C01813=1081.570,6.854,-59.285,174.055,20.252,153.427
C01814=1081.564,6.605,-59.270,174.054,20.250,153.427
C01815=1081.558,6.355,-59.257,174.053,20.248,153.427
C01816=1081.553,6.105,-59.243,174.051,20.245,153.426
C01817=1081.546,5.856,-59.228,174.049,20.243,153.426
C01818=1081.541,5.606,-59.214,174.048,20.241,153.426
C01819=1081.535,5.357,-59.200,174.047,20.239,153.426
C01820=1081.530,5.108,-59.185,174.045,20.237,153.426
C01821=1081.523,4.857,-59.171,174.043,20.235,153.426
C01822=1081.517,4.608,-59.158,174.042,20.233,153.425
C01823=1081.512,4.359,-59.143,174.041,20.231,153.425
C01824=1081.507,4.120,-59.130,174.040,20.229,153.425
C01825=1081.500,3.881,-59.116,174.037,20.226,153.425
C01826=1081.495,3.642,-59.103,174.036,20.224,153.425
C01827=1081.489,3.404,-59.090,174.035,20.222,153.424
C01828=1081.484,3.165,-59.076,174.034,20.220,153.424
C01829=1081.479,2.927,-59.063,174.033,20.218,153.424
C01830=1081.473,2.688,-59.050,174.031,20.216,153.424
C01831=1081.467,2.449,-59.036,174.030,20.214,153.424
C01832=1081.461,2.199,-59.022,174.028,20.211,153.424
C01833=1081.456,1.950,-59.008,174.027,20.209,153.423
C01834=1081.450,1.701,-58.994,174.025,20.207,153.423
C01835=1081.444,1.451,-58.980,174.024,20.205,153.423
C01836=1081.438,1.201,-58.965,174.022,20.203,153.423
C01837=1081.432,0.952,-58.952,174.021,20.201,153.423
C01838=1081.426,0.703,-58.938,174.020,20.198,153.422
C01839=1081.421,0.453,-58.924,174.018,20.196,153.422
C01840=1081.415,0.203,-58.910,174.016,20.194,153.422
C01841=1081.409,-0.047,-58.896,174.015,20.192,153.422
C01842=1081.404,-0.296,-58.882,174.014,20.190,153.422
C01843=1081.398,-0.546,-58.869,174.012,20.188,153.422
C01844=1081.391,-0.822,-58.853,174.010,20.185,153.421
C01845=1081.385,-1.098,-58.837,174.009,20.183,153.421
C01846=1081.378,-1.374,-58.822,174.007,20.180,153.421
C01847=1081.372,-1.650,-58.806,174.006,20.178,153.421
C01848=1081.367,-1.899,-58.792,174.005,20.176,153.421
C01849=1081.360,-2.148,-58.779,174.003,20.173,153.420
C01850=1081.355,-2.398,-58.765,174.001,20.171,153.420
C01851=1081.350,-2.648,-58.751,174.000,20.169,153.420
C01852=1081.344,-2.897,-58.737,173.999,20.167,153.420
C01853=1081.338,-3.146,-58.724,173.997,20.165,153.420
C01854=1081.332,-3.397,-58.710,173.996,20.162,153.420
C01855=1081.326,-3.646,-58.696,173.994,20.160,153.419
C01856=1081.320,-3.896,-58.682,173.993,20.158,153.419
C01857=1081.315,-4.145,-58.669,173.991,20.156,153.419
C01858=1081.308,-4.394,-58.655,173.990,20.154,153.419
C01859=1081.302,-4.645,-58.641,173.988,20.152,153.419
C01860=1081.297,-4.894,-58.627,173.987,20.150,153.419
C01861=1081.290,-5.143,-58.613,173.986,20.148,153.418
C01862=1081.285,-5.392,-58.599,173.984,20.145,153.418
C01863=1081.279,-5.642,-58.586,173.982,20.143,153.418
C01864=1081.273,-5.892,-58.572,173.981,20.141,153.418
C01865=1081.266,-6.141,-58.559,173.980,20.139,153.418
C01866=1081.261,-6.391,-58.545,173.979,20.137,153.418
C01867=1081.255,-6.641,-58.532,173.976,20.135,153.417
C01868=1081.249,-6.890,-58.518,173.975,20.133,153.417
C01869=1081.244,-7.140,-58.504,173.974,20.131,153.417
C01870=1081.237,-7.390,-58.491,173.973,20.129,153.417
C01871=1081.232,-7.639,-58.477,173.971,20.126,153.417
C01872=1081.225,-7.889,-58.464,173.969,20.124,153.417
C01873=1081.220,-8.138,-58.450,173.968,20.122,153.416
C01874=1081.214,-8.388,-58.437,173.967,20.120,153.416
C01875=1081.208,-8.637,-58.423,173.965,20.118,153.416
C01876=1081.202,-8.886,-58.409,173.963,20.116,153.416
C01877=1081.197,-9.136,-58.396,173.962,20.114,153.416
C01878=1081.190,-9.386,-58.382,173.961,20.112,153.416
C01879=1081.184,-9.635,-58.368,173.960,20.110,153.415
C01880=1081.178,-9.885,-58.356,173.957,20.107,153.415
C01881=1081.173,-10.135,-58.342,173.956,20.105,153.415
C01882=1081.167,-10.384,-58.328,173.955,20.103,153.415
C01883=1081.161,-10.634,-58.315,173.954,20.101,153.415
C01884=1081.155,-10.883,-58.301,173.952,20.099,153.415
C01885=1081.150,-11.133,-58.287,173.950,20.097,153.414
C01886=1081.143,-11.382,-58.274,173.949,20.095,153.414
C01887=1081.138,-11.632,-58.261,173.948,20.093,153.414
C01888=1081.132,-11.881,-58.248,173.946,20.091,153.414
C01889=1081.126,-12.131,-58.234,173.945,20.089,153.414
C01890=1081.120,-12.381,-58.220,173.943,20.087,153.414
C01891=1081.114,-12.630,-58.206,173.942,20.085,153.413
C01892=1081.108,-12.880,-58.194,173.940,20.083,153.413
C01893=1081.103,-13.130,-58.180,173.939,20.080,153.413
C01894=1081.097,-13.379,-58.167,173.938,20.078,153.413
C01895=1081.090,-13.628,-58.153,173.936,20.076,153.413
C01896=1081.085,-13.878,-58.139,173.935,20.074,153.413
C01897=1081.079,-14.128,-58.127,173.933,20.072,153.413
C01898=1081.074,-14.377,-58.113,173.932,20.070,153.412
C01899=1081.067,-14.627,-58.100,173.931,20.068,153.412
C01900=1081.062,-14.877,-58.087,173.929,20.065,153.412
C01901=1081.056,-15.126,-58.073,173.928,20.063,153.412
C01902=1081.050,-15.375,-58.060,173.926,20.062,153.412
C01903=1081.044,-15.625,-58.046,173.925,20.060,153.412
C01904=1081.038,-15.875,-58.034,173.924,20.058,153.411
C01905=1081.032,-16.124,-58.020,173.921,20.055,153.411
C01906=1081.027,-16.374,-58.007,173.920,20.053,153.411
C01907=1081.021,-16.624,-57.994,173.919,20.051,153.411
C01908=1081.013,-16.898,-57.979,173.918,20.049,153.411
C01909=1081.008,-17.172,-57.965,173.916,20.047,153.411
C01910=1081.001,-17.447,-57.950,173.914,20.045,153.410
C01911=1080.995,-17.721,-57.936,173.912,20.042,153.410
C01912=1080.989,-17.970,-57.923,173.911,20.040,153.410
C01913=1080.982,-18.220,-57.909,173.910,20.038,153.410
C01914=1080.976,-18.470,-57.897,173.908,20.036,153.410
C01915=1080.971,-18.719,-57.883,173.907,20.034,153.410
C01916=1080.965,-18.968,-57.870,173.905,20.032,153.409
C01917=1080.959,-19.218,-57.857,173.904,20.030,153.409
C01918=1080.953,-19.467,-57.844,173.902,20.028,153.409
C01919=1080.947,-19.717,-57.831,173.901,20.026,153.409
C01920=1080.941,-19.967,-57.817,173.900,20.024,153.409
C01921=1080.935,-20.217,-57.805,173.898,20.021,153.409
C01922=1080.929,-20.466,-57.791,173.897,20.019,153.408
C01923=1080.923,-20.715,-57.778,173.895,20.017,153.408
C01924=1080.918,-20.966,-57.765,173.894,20.015,153.408
C01925=1080.912,-21.215,-57.752,173.892,20.014,153.408
C01926=1080.906,-21.465,-57.739,173.891,20.012,153.408
C01927=1080.899,-21.714,-57.726,173.889,20.009,153.408
C01928=1080.894,-21.964,-57.713,173.888,20.007,153.408
C01929=1080.888,-22.213,-57.700,173.887,20.005,153.407
C01930=1080.882,-22.463,-57.687,173.885,20.003,153.407
C01931=1080.876,-22.713,-57.674,173.884,20.001,153.407
C01932=1080.870,-22.962,-57.661,173.882,19.999,153.407
C01933=1080.865,-23.212,-57.647,173.881,19.997,153.407
C01934=1080.859,-23.462,-57.635,173.879,19.995,153.407
C01935=1080.852,-23.711,-57.621,173.878,19.993,153.406
C01936=1080.847,-23.961,-57.609,173.877,19.991,153.406
C01937=1080.841,-24.210,-57.596,173.875,19.989,153.406
C01938=1080.835,-24.459,-57.583,173.873,19.987,153.406
C01939=1080.830,-24.709,-57.570,173.872,19.985,153.406
C01940=1080.824,-24.959,-57.557,173.871,19.983,153.406
C01941=1080.818,-25.209,-57.545,173.869,19.981,153.406
C01942=1080.811,-25.458,-57.531,173.868,19.979,153.405
C01943=1080.806,-25.708,-57.519,173.866,19.976,153.405
C01944=1080.799,-25.957,-57.505,173.865,19.974,153.405
C01945=1080.794,-26.207,-57.492,173.864,19.972,153.405
C01946=1080.789,-26.457,-57.480,173.862,19.970,153.405
C01947=1080.783,-26.706,-57.467,173.861,19.968,153.405
C01948=1080.777,-26.956,-57.454,173.860,19.967,153.405
C01949=1080.771,-27.205,-57.441,173.857,19.964,153.405
C01950=1080.765,-27.455,-57.428,173.856,19.962,153.404
C01951=1080.759,-27.705,-57.416,173.855,19.960,153.404
C01952=1080.753,-27.954,-57.403,173.854,19.958,153.404
C01953=1080.747,-28.204,-57.390,173.852,19.957,153.404
C01954=1080.741,-28.454,-57.378,173.851,19.955,153.404
C01955=1080.734,-28.703,-57.364,173.849,19.952,153.404
C01956=1080.729,-28.953,-57.352,173.848,19.950,153.404
C01957=1080.723,-29.202,-57.339,173.846,19.948,153.403
C01958=1080.717,-29.451,-57.326,173.845,19.947,153.403
C01959=1080.711,-29.701,-57.314,173.844,19.945,153.403
C01960=1080.705,-29.951,-57.301,173.842,19.943,153.403
C01961=1080.699,-30.201,-57.289,173.840,19.940,153.403
C01962=1080.693,-30.450,-57.275,173.839,19.938,153.403
C01963=1080.687,-30.700,-57.263,173.837,19.937,153.403
C01964=1080.681,-30.950,-57.250,173.836,19.935,153.402
C01965=1080.676,-31.199,-57.238,173.835,19.933,153.402
C01966=1080.669,-31.448,-57.225,173.834,19.931,153.402
C01967=1080.663,-31.698,-57.213,173.832,19.929,153.402
C01968=1080.657,-31.948,-57.200,173.830,19.927,153.402
C01969=1080.651,-32.198,-57.188,173.829,19.925,153.402
C01970=1080.645,-32.447,-57.174,173.827,19.923,153.402
C01971=1080.639,-32.697,-57.162,173.826,19.921,153.401
C01972=1080.633,-32.970,-57.148,173.825,19.919,153.401
C01973=1080.627,-33.244,-57.134,173.823,19.916,153.401
C01974=1080.620,-33.517,-57.121,173.822,19.914,153.401
C01975=1080.613,-33.791,-57.107,173.819,19.912,153.401
C01976=1080.608,-34.041,-57.094,173.818,19.910,153.401
C01977=1080.602,-34.290,-57.082,173.817,19.908,153.401
C01978=1080.596,-34.540,-57.070,173.815,19.906,153.401
C01979=1080.590,-34.790,-57.057,173.814,19.904,153.400
C01980=1080.584,-35.039,-57.044,173.813,19.903,153.400
C01981=1080.578,-35.289,-57.031,173.811,19.901,153.400
C01982=1080.572,-35.539,-57.019,173.809,19.898,153.400
C01983=1080.566,-35.787,-57.007,173.808,19.896,153.400
C01984=1080.560,-36.037,-56.994,173.807,19.894,153.400
C01985=1080.555,-36.287,-56.982,173.805,19.893,153.400
C01986=1080.549,-36.537,-56.969,173.804,19.891,153.399
C01987=1080.543,-36.786,-56.957,173.803,19.889,153.399
C01988=1080.537,-37.036,-56.945,173.802,19.887,153.399
C01989=1080.532,-37.286,-56.932,173.799,19.885,153.399
C01990=1080.525,-37.535,-56.919,173.798,19.883,153.399
C01991=1080.519,-37.784,-56.907,173.797,19.881,153.399
C01992=1080.513,-38.034,-56.895,173.795,19.879,153.399
C01993=1080.507,-38.284,-56.882,173.794,19.877,153.399
C01994=1080.502,-38.534,-56.870,173.793,19.875,153.398
C01995=1080.496,-38.783,-56.857,173.791,19.873,153.398
C01996=1080.490,-39.033,-56.845,173.789,19.871,153.398
C01997=1080.484,-39.282,-56.833,173.788,19.869,153.398
C01998=1080.478,-39.532,-56.820,173.787,19.867,153.398
C01999=1080.472,-39.782,-56.808,173.785,19.866,153.398
C02000=1080.466,-40.031,-56.796,173.784,19.864,153.398
C02001=1080.460,-40.281,-56.784,173.783,19.862,153.398
C02002=1080.454,-40.531,-56.771,173.781,19.860,153.398
C02003=1080.447,-40.780,-56.759,173.779,19.858,153.397
C02004=1080.442,-41.030,-56.747,173.778,19.856,153.397
C02005=1080.436,-41.280,-56.734,173.776,19.854,153.397
C02006=1080.429,-41.529,-56.722,173.775,19.852,153.397
C02007=1080.424,-41.779,-56.710,173.774,19.850,153.397
C02008=1080.418,-42.028,-56.698,173.772,19.849,153.397
C02009=1080.412,-42.278,-56.686,173.771,19.847,153.397
C02010=1080.406,-42.528,-56.673,173.770,19.845,153.397
C02011=1080.401,-42.777,-56.662,173.767,19.843,153.397
C02012=1080.394,-43.027,-56.650,173.766,19.841,153.396
C02013=1080.388,-43.277,-56.637,173.765,19.839,153.396
C02014=1080.382,-43.527,-56.625,173.763,19.837,153.396
C02015=1080.376,-43.776,-56.613,173.762,19.835,153.396
C02016=1080.370,-44.025,-56.600,173.761,19.834,153.396
C02017=1080.364,-44.275,-56.588,173.759,19.832,153.396
C02018=1080.358,-44.524,-56.576,173.758,19.830,153.396
C02019=1080.352,-44.774,-56.564,173.756,19.828,153.396
C02020=1080.347,-45.025,-56.552,173.755,19.826,153.395
C02021=1080.341,-45.274,-56.540,173.753,19.824,153.395
C02022=1080.335,-45.523,-56.528,173.752,19.822,153.395
C02023=1080.329,-45.773,-56.515,173.751,19.820,153.395
C02024=1080.323,-46.022,-56.504,173.749,19.819,153.395
C02025=1080.317,-46.272,-56.491,173.748,19.817,153.395
C02026=1080.311,-46.522,-56.480,173.746,19.815,153.395
C02027=1080.305,-46.771,-56.468,173.745,19.813,153.395
C02028=1080.299,-47.021,-56.455,173.743,19.811,153.395
C02029=1080.293,-47.271,-56.443,173.742,19.809,153.395
C02030=1080.287,-47.520,-56.431,173.740,19.807,153.394
C02031=1080.281,-47.770,-56.420,173.739,19.806,153.394
C02032=1080.275,-48.020,-56.407,173.738,19.804,153.394
C02033=1080.270,-48.269,-56.395,173.736,19.802,153.394
C02034=1080.263,-48.519,-56.383,173.735,19.800,153.394
C02035=1080.258,-48.769,-56.372,173.734,19.798,153.394
C02036=1080.251,-49.042,-56.358,173.731,19.796,153.394
C02037=1080.245,-49.316,-56.344,173.730,19.794,153.394
C02038=1080.238,-49.590,-56.332,173.729,19.792,153.393
C02039=1080.232,-49.864,-56.318,173.727,19.790,153.393
C02040=1080.225,-50.114,-56.307,173.725,19.788,153.393
C02041=1080.220,-50.363,-56.295,173.724,19.786,153.393
C02042=1080.214,-50.613,-56.283,173.722,19.785,153.393
C02043=1080.208,-50.863,-56.271,173.721,19.783,153.393
C02044=1080.202,-51.112,-56.259,173.720,19.781,153.393
C02045=1080.195,-51.362,-56.247,173.718,19.779,153.393
C02046=1080.190,-51.612,-56.236,173.717,19.778,153.393
C02047=1080.184,-51.861,-56.224,173.715,19.776,153.393
C02048=1080.177,-52.111,-56.212,173.713,19.774,153.393
C02049=1080.171,-52.361,-56.200,173.712,19.772,153.393
C02050=1080.165,-52.610,-56.189,173.711,19.770,153.392
C02051=1080.159,-52.860,-56.177,173.709,19.769,153.392
C02052=1080.153,-53.110,-56.165,173.708,19.767,153.392
C02053=1080.147,-53.359,-56.153,173.706,19.765,153.392
C02054=1080.140,-53.609,-56.141,173.705,19.764,153.392
C02055=1080.135,-53.859,-56.130,173.704,19.762,153.392
C02056=1080.129,-54.108,-56.118,173.702,19.760,153.392
C02057=1080.122,-54.358,-56.107,173.701,19.759,153.392
C02058=1080.117,-54.607,-56.094,173.699,19.757,153.392
C02059=1080.110,-54.857,-56.082,173.698,19.755,153.392
C02060=1080.104,-55.107,-56.071,173.696,19.753,153.392
C02061=1080.098,-55.356,-56.060,173.694,19.751,153.392
C02062=1080.092,-55.607,-56.048,173.693,19.750,153.392
C02063=1080.086,-55.855,-56.036,173.692,19.748,153.391
C02064=1080.080,-56.106,-56.025,173.690,19.746,153.391
C02065=1080.074,-56.356,-56.012,173.689,19.744,153.391
C02066=1080.068,-56.604,-56.001,173.687,19.743,153.391
C02067=1080.062,-56.855,-55.990,173.686,19.741,153.391
C02068=1080.056,-57.103,-55.978,173.685,19.739,153.391
C02069=1080.050,-57.354,-55.966,173.683,19.738,153.391
C02070=1080.044,-57.603,-55.954,173.682,19.736,153.391
C02071=1080.038,-57.853,-55.943,173.680,19.734,153.391
C02072=1080.031,-58.103,-55.931,173.678,19.732,153.391
C02073=1080.026,-58.352,-55.920,173.677,19.730,153.391
C02074=1080.019,-58.602,-55.908,173.675,19.729,153.391
C02075=1080.014,-58.851,-55.897,173.674,19.727,153.391
C02076=1080.007,-59.102,-55.886,173.673,19.725,153.390
C02077=1080.002,-59.351,-55.874,173.671,19.724,153.390
C02078=1079.996,-59.601,-55.862,173.670,19.722,153.390
C02079=1079.990,-59.850,-55.851,173.668,19.720,153.390
C02080=1079.983,-60.100,-55.839,173.667,19.719,153.390
C02081=1079.978,-60.349,-55.827,173.665,19.717,153.390
C02082=1079.972,-60.599,-55.816,173.664,19.715,153.390
C02083=1079.966,-60.848,-55.804,173.663,19.714,153.390
C02084=1079.959,-61.099,-55.793,173.661,19.712,153.390
C02085=1079.954,-61.348,-55.782,173.660,19.710,153.390
C02086=1079.948,-61.598,-55.770,173.658,19.708,153.390
C02087=1079.942,-61.847,-55.759,173.656,19.707,153.390
C02088=1079.935,-62.097,-55.747,173.655,19.705,153.389
C02089=1079.930,-62.346,-55.736,173.653,19.703,153.389
C02090=1079.924,-62.597,-55.724,173.652,19.702,153.389
C02091=1079.918,-62.846,-55.713,173.651,19.700,153.389
C02092=1079.912,-63.096,-55.701,173.649,19.698,153.389
C02093=1079.906,-63.346,-55.690,173.648,19.697,153.389
C02094=1079.899,-63.595,-55.679,173.646,19.695,153.389
C02095=1079.894,-63.845,-55.667,173.645,19.693,153.389
C02096=1079.888,-64.095,-55.656,173.644,19.692,153.389
C02097=1079.882,-64.344,-55.644,173.642,19.690,153.389
C02098=1079.875,-64.594,-55.633,173.641,19.688,153.389
C02099=1079.870,-64.844,-55.622,173.639,19.687,153.389
C02100=1079.864,-65.118,-55.609,173.637,19.685,153.389
C02101=1079.856,-65.394,-55.597,173.636,19.683,153.389
C02102=1079.850,-65.669,-55.584,173.634,19.681,153.389
C02103=1079.843,-65.945,-55.572,173.633,19.680,153.389
C02104=1079.837,-66.194,-55.560,173.632,19.678,153.388
C02105=1079.832,-66.444,-55.549,173.630,19.676,153.388
C02106=1079.826,-66.694,-55.538,173.629,19.675,153.388
C02107=1079.820,-66.943,-55.527,173.627,19.672,153.388
C02108=1079.813,-67.193,-55.515,173.625,19.671,153.388
C02109=1079.808,-67.442,-55.504,173.624,19.669,153.388
C02110=1079.802,-67.692,-55.493,173.622,19.668,153.388
C02111=1079.796,-67.942,-55.482,173.621,19.666,153.388
C02112=1079.790,-68.191,-55.470,173.619,19.664,153.388
C02113=1079.784,-68.441,-55.458,173.618,19.663,153.388
C02114=1079.778,-68.691,-55.448,173.616,19.661,153.388
C02115=1079.773,-68.940,-55.437,173.615,19.659,153.388
C02116=1079.766,-69.190,-55.425,173.614,19.658,153.388
C02117=1079.760,-69.439,-55.414,173.612,19.656,153.388
C02118=1079.754,-69.689,-55.403,173.611,19.655,153.388
C02119=1079.748,-69.939,-55.392,173.609,19.653,153.388
C02120=1079.743,-70.189,-55.380,173.608,19.651,153.387
C02121=1079.737,-70.438,-55.369,173.606,19.650,153.387
C02122=1079.731,-70.689,-55.358,173.605,19.648,153.387
C02123=1079.725,-70.938,-55.347,173.604,19.647,153.387
C02124=1079.719,-71.187,-55.336,173.602,19.645,153.387
C02125=1079.713,-71.437,-55.324,173.601,19.643,153.387
C02126=1079.707,-71.687,-55.313,173.599,19.642,153.387
C02127=1079.701,-71.936,-55.303,173.598,19.640,153.387
C02128=1079.695,-72.186,-55.291,173.596,19.639,153.387
C02129=1079.690,-72.436,-55.280,173.595,19.637,153.387
C02130=1079.684,-72.686,-55.269,173.594,19.635,153.387
C02131=1079.678,-72.936,-55.258,173.592,19.634,153.387
C02132=1079.672,-73.185,-55.247,173.591,19.632,153.387
C02133=1079.666,-73.435,-55.236,173.589,19.631,153.387
C02134=1079.660,-73.685,-55.225,173.588,19.629,153.387
C02135=1079.654,-73.934,-55.214,173.585,19.627,153.387
C02136=1079.648,-74.183,-55.202,173.584,19.625,153.387
C02137=1079.643,-74.433,-55.191,173.583,19.624,153.387
C02138=1079.636,-74.683,-55.180,173.581,19.622,153.387
C02139=1079.631,-74.932,-55.169,173.580,19.621,153.387
C02140=1079.624,-75.183,-55.158,173.578,19.619,153.387
C02141=1079.618,-75.432,-55.148,173.577,19.618,153.386
C02142=1079.612,-75.681,-55.137,173.575,19.616,153.386
C02143=1079.606,-75.931,-55.126,173.574,19.615,153.386
C02144=1079.600,-76.181,-55.115,173.572,19.613,153.386
C02145=1079.594,-76.430,-55.104,173.571,19.612,153.386
C02146=1079.588,-76.681,-55.093,173.569,19.610,153.386
C02147=1079.582,-76.930,-55.082,173.568,19.609,153.386
C02148=1079.576,-77.180,-55.071,173.566,19.607,153.386
C02149=1079.570,-77.429,-55.061,173.565,19.606,153.386
C02150=1079.564,-77.679,-55.049,173.563,19.604,153.386
C02151=1079.558,-77.928,-55.039,173.562,19.603,153.386
C02152=1079.552,-78.179,-55.028,173.560,19.601,153.386
C02153=1079.546,-78.429,-55.017,173.559,19.600,153.386
C02154=1079.540,-78.678,-55.006,173.558,19.598,153.386
C02155=1079.535,-78.928,-54.995,173.556,19.597,153.386
C02156=1079.528,-79.177,-54.985,173.555,19.595,153.386
C02157=1079.522,-79.427,-54.974,173.553,19.594,153.386
C02158=1079.516,-79.677,-54.963,173.552,19.592,153.386
C02159=1079.510,-79.926,-54.952,173.550,19.591,153.386
C02160=1079.504,-80.176,-54.941,173.549,19.589,153.386
C02161=1079.497,-80.425,-54.931,173.547,19.588,153.386
C02162=1079.492,-80.675,-54.920,173.546,19.586,153.386
C02163=1079.486,-80.926,-54.909,173.544,19.585,153.386
C02164=1079.479,-81.202,-54.898,173.543,19.584,153.386
C02165=1079.472,-81.480,-54.886,173.541,19.582,153.386
C02166=1079.466,-81.757,-54.873,173.540,19.581,153.386
C02167=1079.458,-82.034,-54.861,173.537,19.579,153.386
C02168=1079.453,-82.284,-54.851,173.537,19.578,153.386
C02169=1079.446,-82.535,-54.840,173.535,19.577,153.386
C02170=1079.440,-82.784,-54.830,173.534,19.575,153.386
C02171=1079.434,-83.033,-54.819,173.532,19.574,153.386
C02172=1079.428,-83.282,-54.809,173.531,19.572,153.386
C02173=1079.422,-83.533,-54.798,173.529,19.571,153.386
C02174=1079.416,-83.783,-54.787,173.528,19.570,153.386
C02175=1079.409,-84.032,-54.777,173.526,19.568,153.386
C02176=1079.403,-84.282,-54.766,173.525,19.567,153.386
C02177=1079.397,-84.532,-54.755,173.523,19.565,153.386
C02178=1079.391,-84.781,-54.745,173.522,19.564,153.386
C02179=1079.385,-85.031,-54.734,173.520,19.562,153.386
C02180=1079.379,-85.281,-54.723,173.518,19.561,153.386
C02181=1079.373,-85.530,-54.713,173.517,19.560,153.386
C02182=1079.367,-85.780,-54.703,173.515,19.558,153.386
C02183=1079.361,-86.030,-54.692,173.514,19.557,153.386
C02184=1079.354,-86.280,-54.681,173.513,19.555,153.386
C02185=1079.349,-86.529,-54.670,173.511,19.554,153.386
C02186=1079.342,-86.779,-54.661,173.509,19.553,153.386
C02187=1079.337,-87.029,-54.650,173.508,19.551,153.386
C02188=1079.330,-87.278,-54.640,173.506,19.550,153.386
C02189=1079.324,-87.529,-54.629,173.505,19.549,153.386
C02190=1079.318,-87.778,-54.618,173.503,19.547,153.386
C02191=1079.312,-88.027,-54.608,173.502,19.546,153.386
C02192=1079.306,-88.277,-54.598,173.500,19.544,153.386
C02193=1079.300,-88.527,-54.587,173.499,19.543,153.386
C02194=1079.294,-88.777,-54.576,173.497,19.542,153.386
C02195=1079.288,-89.027,-54.566,173.496,19.540,153.386
C02196=1079.282,-89.276,-54.556,173.494,19.539,153.386
C02197=1079.276,-89.525,-54.545,173.493,19.537,153.386
C02198=1079.270,-89.775,-54.535,173.491,19.536,153.386
C02199=1079.264,-90.025,-54.524,173.489,19.535,153.386
C02200=1079.258,-90.275,-54.513,173.489,19.534,153.386
C02201=1079.252,-90.525,-54.504,173.487,19.532,153.386
C02202=1079.246,-90.774,-54.493,173.486,19.532,153.386
C02203=1079.240,-91.024,-54.483,173.484,19.530,153.386
C02204=1079.234,-91.274,-54.472,173.483,19.529,153.386
C02205=1079.227,-91.523,-54.462,173.481,19.528,153.386
C02206=1079.221,-91.774,-54.451,173.479,19.526,153.386
C02207=1079.215,-92.023,-54.441,173.478,19.525,153.386
C02208=1079.210,-92.273,-54.431,173.476,19.524,153.386
C02209=1079.204,-92.522,-54.420,173.475,19.522,153.386
C02210=1079.198,-92.772,-54.411,173.473,19.521,153.386
C02211=1079.192,-93.022,-54.400,173.472,19.519,153.386
C02212=1079.185,-93.271,-54.389,173.470,19.518,153.386
C02213=1079.180,-93.521,-54.379,173.469,19.517,153.386
C02214=1079.173,-93.770,-54.369,173.467,19.515,153.386
C02215=1079.167,-94.021,-54.358,173.465,19.514,153.386
C02216=1079.161,-94.270,-54.348,173.464,19.513,153.386
C02217=1079.156,-94.520,-54.338,173.463,19.511,153.386
C02218=1079.149,-94.769,-54.328,173.462,19.511,153.386
C02219=1079.144,-95.019,-54.318,173.460,19.509,153.386
C02220=1079.137,-95.269,-54.307,173.459,19.508,153.386
C02221=1079.132,-95.519,-54.297,173.457,19.507,153.386
C02222=1079.125,-95.768,-54.287,173.456,19.505,153.386
C02223=1079.120,-96.018,-54.277,173.454,19.504,153.386
C02224=1079.114,-96.268,-54.267,173.452,19.503,153.386
C02225=1079.108,-96.517,-54.256,173.451,19.501,153.386
C02226=1079.102,-96.767,-54.247,173.449,19.500,153.386
C02227=1079.096,-97.017,-54.236,173.448,19.499,153.386
C02228=1079.089,-97.297,-54.224,173.446,19.497,153.386
C02229=1079.082,-97.576,-54.213,173.444,19.496,153.386
C02230=1079.076,-97.856,-54.202,173.443,19.495,153.386
C02231=1079.068,-98.136,-54.190,173.442,19.493,153.386
C02232=1079.062,-98.386,-54.180,173.440,19.493,153.387
C02233=1079.056,-98.635,-54.170,173.438,19.491,153.387
C02234=1079.050,-98.885,-54.160,173.437,19.490,153.387
C02235=1079.044,-99.135,-54.150,173.435,19.489,153.387
C02236=1079.038,-99.384,-54.140,173.433,19.488,153.387
C02237=1079.032,-99.634,-54.130,173.432,19.487,153.387
C02238=1079.026,-99.883,-54.120,173.430,19.485,153.387
C02239=1079.020,-100.133,-54.110,173.429,19.484,153.387
C02240=1079.014,-100.383,-54.100,173.427,19.483,153.387
C02241=1079.007,-100.632,-54.090,173.425,19.482,153.387
C02242=1079.001,-100.882,-54.080,173.424,19.480,153.387
C02243=1078.996,-101.132,-54.070,173.423,19.480,153.387
C02244=1078.989,-101.382,-54.059,173.422,19.478,153.387
C02245=1078.983,-101.632,-54.050,173.420,19.477,153.387
C02246=1078.977,-101.882,-54.040,173.418,19.476,153.387
C02247=1078.971,-102.131,-54.029,173.417,19.475,153.387
C02248=1078.965,-102.381,-54.020,173.415,19.473,153.387
C02249=1078.958,-102.631,-54.010,173.413,19.472,153.387
C02250=1078.953,-102.881,-54.000,173.412,19.471,153.387
C02251=1078.946,-103.130,-53.990,173.410,19.470,153.387
C02252=1078.940,-103.380,-53.980,173.409,19.469,153.388
C02253=1078.935,-103.630,-53.970,173.408,19.468,153.387
C02254=1078.928,-103.879,-53.960,173.406,19.467,153.388
C02255=1078.922,-104.129,-53.950,173.405,19.466,153.388
C02256=1078.916,-104.379,-53.941,173.403,19.465,153.388
C02257=1078.911,-104.629,-53.930,173.401,19.464,153.388
C02258=1078.904,-104.878,-53.920,173.400,19.462,153.388
C02259=1078.898,-105.128,-53.911,173.398,19.461,153.388
C02260=1078.892,-105.378,-53.901,173.396,19.460,153.388
C02261=1078.886,-105.628,-53.891,173.395,19.459,153.388
C02262=1078.880,-105.877,-53.881,173.394,19.458,153.388
C02263=1078.874,-106.127,-53.871,173.392,19.457,153.388
C02264=1078.867,-106.376,-53.861,173.391,19.456,153.388
C02265=1078.861,-106.626,-53.852,173.389,19.455,153.388
C02266=1078.856,-106.876,-53.842,173.388,19.454,153.388
C02267=1078.850,-107.126,-53.832,173.386,19.452,153.388
C02268=1078.843,-107.375,-53.822,173.384,19.451,153.388
C02269=1078.837,-107.625,-53.812,173.383,19.450,153.389
C02270=1078.831,-107.875,-53.803,173.382,19.449,153.389
C02271=1078.825,-108.125,-53.793,173.380,19.448,153.389
C02272=1078.819,-108.374,-53.784,173.379,19.447,153.389
C02273=1078.813,-108.625,-53.773,173.377,19.447,153.389
C02274=1078.807,-108.874,-53.763,173.375,19.445,153.389
C02275=1078.800,-109.124,-53.754,173.374,19.444,153.389
C02276=1078.794,-109.373,-53.744,173.372,19.443,153.389
C02277=1078.788,-109.623,-53.734,173.370,19.442,153.389
C02278=1078.782,-109.873,-53.725,173.370,19.441,153.389
C02279=1078.776,-110.123,-53.715,173.368,19.440,153.389
C02280=1078.770,-110.373,-53.706,173.366,19.439,153.389
C02281=1078.763,-110.622,-53.696,173.364,19.438,153.389
C02282=1078.757,-110.872,-53.687,173.363,19.437,153.390
C02283=1078.751,-111.121,-53.677,173.361,19.436,153.390
C02284=1078.745,-111.370,-53.667,173.360,19.435,153.390
C02285=1078.740,-111.621,-53.657,173.359,19.434,153.390
C02286=1078.734,-111.870,-53.647,173.357,19.433,153.390
C02287=1078.727,-112.120,-53.638,173.355,19.432,153.390
C02288=1078.721,-112.370,-53.628,173.354,19.431,153.390
C02289=1078.715,-112.620,-53.619,173.352,19.430,153.390
C02290=1078.709,-112.870,-53.609,173.350,19.429,153.390
C02291=1078.703,-113.119,-53.600,173.349,19.428,153.390
C02292=1078.696,-113.396,-53.589,173.347,19.427,153.390
C02293=1078.689,-113.673,-53.579,173.346,19.426,153.390
C02294=1078.682,-113.950,-53.568,173.344,19.425,153.391
C02295=1078.676,-114.227,-53.557,173.342,19.424,153.391
C02296=1078.670,-114.476,-53.548,173.340,19.423,153.391
C02297=1078.664,-114.726,-53.538,173.340,19.422,153.391
C02298=1078.658,-114.975,-53.529,173.338,19.421,153.391
C02299=1078.652,-115.225,-53.519,173.336,19.420,153.391
C02300=1078.645,-115.475,-53.509,173.334,19.419,153.391
C02301=1078.639,-115.724,-53.501,173.333,19.418,153.391
C02302=1078.632,-115.974,-53.491,173.331,19.417,153.391
C02303=1078.626,-116.224,-53.481,173.330,19.416,153.391
C02304=1078.620,-116.474,-53.472,173.329,19.415,153.391
C02305=1078.614,-116.724,-53.462,173.327,19.415,153.392
C02306=1078.608,-116.973,-53.453,173.325,19.414,153.392
C02307=1078.602,-117.222,-53.443,173.323,19.413,153.392
C02308=1078.596,-117.472,-53.434,173.322,19.412,153.392
C02309=1078.590,-117.723,-53.425,173.321,19.411,153.392
C02310=1078.584,-117.973,-53.415,173.319,19.410,153.392
C02311=1078.578,-118.222,-53.406,173.318,19.409,153.392
C02312=1078.572,-118.472,-53.396,173.316,19.408,153.392
C02313=1078.565,-118.722,-53.387,173.314,19.407,153.392
C02314=1078.559,-118.972,-53.377,173.312,19.406,153.393
C02315=1078.553,-119.220,-53.369,173.312,19.406,153.393
C02316=1078.547,-119.470,-53.359,173.310,19.405,153.393
C02317=1078.541,-119.720,-53.349,173.308,19.404,153.393
C02318=1078.535,-119.971,-53.341,173.306,19.403,153.393
C02319=1078.529,-120.220,-53.331,173.305,19.402,153.393
C02320=1078.522,-120.470,-53.322,173.303,19.401,153.393
C02321=1078.516,-120.720,-53.312,173.302,19.401,153.393
C02322=1078.511,-120.969,-53.303,173.300,19.400,153.393
C02323=1078.504,-121.218,-53.294,173.299,19.399,153.394
C02324=1078.498,-121.469,-53.285,173.297,19.398,153.394
C02325=1078.492,-121.719,-53.275,173.295,19.397,153.394
C02326=1078.485,-121.969,-53.266,173.294,19.396,153.394
C02327=1078.479,-122.218,-53.256,173.293,19.395,153.394
C02328=1078.474,-122.467,-53.247,173.291,19.394,153.394
C02329=1078.468,-122.718,-53.238,173.289,19.394,153.394
C02330=1078.461,-122.967,-53.229,173.287,19.393,153.394
C02331=1078.455,-123.217,-53.220,173.286,19.393,153.395
C02332=1078.449,-123.467,-53.210,173.285,19.392,153.395
C02333=1078.442,-123.717,-53.200,173.283,19.391,153.395
C02334=1078.437,-123.966,-53.192,173.281,19.390,153.395
C02335=1078.430,-124.216,-53.183,173.280,19.389,153.395
C02336=1078.424,-124.466,-53.173,173.279,19.388,153.395
C02337=1078.418,-124.715,-53.164,173.277,19.387,153.395
C02338=1078.412,-124.966,-53.155,173.275,19.387,153.395
C02339=1078.406,-125.215,-53.146,173.273,19.386,153.396
C02340=1078.400,-125.464,-53.137,173.272,19.385,153.396
C02341=1078.394,-125.715,-53.128,173.271,19.384,153.396
C02342=1078.388,-125.965,-53.118,173.269,19.383,153.396
C02343=1078.381,-126.214,-53.109,173.267,19.383,153.396
C02344=1078.375,-126.463,-53.100,173.265,19.382,153.396
C02345=1078.369,-126.714,-53.091,173.264,19.381,153.396
C02346=1078.363,-126.964,-53.082,173.263,19.381,153.396
C02347=1078.356,-127.213,-53.073,173.261,19.380,153.397
C02348=1078.350,-127.463,-53.064,173.259,19.379,153.397
C02349=1078.344,-127.713,-53.054,173.257,19.378,153.397
C02350=1078.338,-127.964,-53.046,173.257,19.378,153.397
C02351=1078.334,-128.214,-53.037,173.255,19.376,153.397
C02352=1078.332,-128.468,-53.025,173.254,19.374,153.397
C02353=1078.334,-128.722,-53.012,173.253,19.371,153.396
C02354=1078.338,-128.975,-53.000,173.253,19.367,153.396
C02355=1078.346,-129.226,-52.986,173.253,19.362,153.395
C02356=1077.949,-129.248,-53.132,173.208,19.486,153.425
C02357=1077.941,-128.998,-53.147,173.209,19.491,153.426
C02358=1077.936,-128.745,-53.159,173.209,19.496,153.427
C02359=1077.935,-128.490,-53.172,173.210,19.499,153.427
C02360=1077.936,-128.235,-53.183,173.211,19.501,153.428
C02361=1077.940,-127.986,-53.193,173.211,19.502,153.428
C02362=1077.946,-127.735,-53.202,173.213,19.503,153.428
C02363=1077.952,-127.485,-53.211,173.215,19.504,153.428
C02364=1077.959,-127.235,-53.220,173.217,19.505,153.427
C02365=1077.965,-126.986,-53.229,173.218,19.506,153.427
C02366=1077.971,-126.735,-53.238,173.219,19.506,153.427
C02367=1077.977,-126.486,-53.247,173.221,19.507,153.427
C02368=1077.983,-126.237,-53.256,173.223,19.508,153.427
C02369=1077.989,-125.986,-53.265,173.224,19.509,153.427
C02370=1077.995,-125.736,-53.275,173.226,19.509,153.427
C02371=1078.002,-125.487,-53.284,173.227,19.510,153.427
C02372=1078.008,-125.237,-53.292,173.229,19.511,153.426
C02373=1078.014,-124.987,-53.302,173.231,19.512,153.426
C02374=1078.020,-124.738,-53.311,173.232,19.513,153.426
C02375=1078.027,-124.488,-53.320,173.234,19.514,153.426
C02376=1078.033,-124.238,-53.329,173.235,19.514,153.426
C02377=1078.039,-123.988,-53.339,173.237,19.514,153.426
C02378=1078.045,-123.739,-53.348,173.239,19.515,153.426
C02379=1078.051,-123.489,-53.358,173.240,19.516,153.425
C02380=1078.057,-123.239,-53.366,173.242,19.517,153.425
C02381=1078.063,-122.989,-53.375,173.243,19.518,153.425
C02382=1078.070,-122.739,-53.385,173.245,19.519,153.425
C02383=1078.075,-122.490,-53.394,173.246,19.520,153.425
C02384=1078.081,-122.240,-53.404,173.248,19.521,153.425
C02385=1078.087,-121.990,-53.413,173.250,19.522,153.425
C02386=1078.094,-121.740,-53.422,173.251,19.522,153.425
C02387=1078.100,-121.491,-53.431,173.252,19.523,153.425
C02388=1078.106,-121.241,-53.441,173.254,19.524,153.425
C02389=1078.112,-120.992,-53.450,173.256,19.525,153.424
C02390=1078.118,-120.742,-53.460,173.257,19.526,153.424
C02391=1078.124,-120.492,-53.468,173.259,19.527,153.424
C02392=1078.130,-120.242,-53.478,173.260,19.527,153.424
C02393=1078.137,-119.992,-53.487,173.262,19.528,153.424
C02394=1078.143,-119.742,-53.496,173.263,19.529,153.424
C02395=1078.150,-119.493,-53.506,173.265,19.530,153.424
C02396=1078.155,-119.244,-53.515,173.267,19.531,153.424
C02397=1078.161,-118.994,-53.525,173.268,19.532,153.424
C02398=1078.167,-118.743,-53.534,173.269,19.533,153.423
C02399=1078.173,-118.494,-53.543,173.271,19.534,153.423
C02400=1078.179,-118.244,-53.553,173.273,19.534,153.423
C02401=1078.186,-117.994,-53.562,173.275,19.535,153.423
C02402=1078.192,-117.744,-53.572,173.276,19.536,153.423
C02403=1078.199,-117.495,-53.581,173.277,19.537,153.423
C02404=1078.204,-117.246,-53.590,173.279,19.538,153.423
C02405=1078.210,-116.996,-53.600,173.281,19.539,153.423
C02406=1078.217,-116.746,-53.609,173.282,19.540,153.423
C02407=1078.223,-116.496,-53.619,173.284,19.541,153.422
C02408=1078.229,-116.246,-53.628,173.286,19.542,153.422
C02409=1078.235,-115.997,-53.638,173.287,19.542,153.422
C02410=1078.241,-115.747,-53.648,173.288,19.544,153.422
C02411=1078.247,-115.497,-53.657,173.290,19.545,153.422
C02412=1078.254,-115.247,-53.667,173.292,19.545,153.422
C02413=1078.260,-114.997,-53.676,173.293,19.546,153.422
C02414=1078.266,-114.747,-53.685,173.295,19.547,153.422
C02415=1078.271,-114.498,-53.694,173.297,19.548,153.422
C02416=1078.277,-114.248,-53.704,173.298,19.549,153.422
C02417=1078.284,-113.971,-53.715,173.299,19.550,153.421
C02418=1078.291,-113.695,-53.725,173.302,19.552,153.421
C02419=1078.298,-113.418,-53.736,173.303,19.553,153.421
C02420=1078.305,-113.141,-53.746,173.305,19.554,153.421
C02421=1078.311,-112.891,-53.756,173.306,19.554,153.421
C02422=1078.317,-112.641,-53.766,173.308,19.555,153.421
C02423=1078.323,-112.391,-53.775,173.309,19.557,153.421
C02424=1078.329,-112.142,-53.785,173.311,19.558,153.421
C02425=1078.335,-111.892,-53.794,173.312,19.558,153.421
C02426=1078.342,-111.642,-53.804,173.314,19.559,153.421
C02427=1078.348,-111.393,-53.814,173.316,19.560,153.421
C02428=1078.354,-111.143,-53.824,173.317,19.562,153.421
C02429=1078.360,-110.893,-53.833,173.318,19.562,153.421
C02430=1078.366,-110.643,-53.843,173.320,19.563,153.420
C02431=1078.372,-110.393,-53.853,173.322,19.564,153.420
C02432=1078.378,-110.143,-53.863,173.323,19.566,153.420
C02433=1078.384,-109.894,-53.872,173.325,19.567,153.420
C02434=1078.390,-109.644,-53.882,173.327,19.568,153.420
C02435=1078.397,-109.394,-53.891,173.328,19.569,153.420
C02436=1078.403,-109.144,-53.901,173.329,19.570,153.420
C02437=1078.409,-108.895,-53.911,173.331,19.571,153.420
C02438=1078.415,-108.645,-53.921,173.332,19.572,153.420
C02439=1078.422,-108.396,-53.930,173.334,19.573,153.420
C02440=1078.428,-108.146,-53.940,173.336,19.574,153.420
C02441=1078.433,-107.896,-53.950,173.337,19.575,153.420
C02442=1078.439,-107.646,-53.960,173.339,19.576,153.419
C02443=1078.446,-107.397,-53.970,173.340,19.577,153.420
C02444=1078.452,-107.147,-53.979,173.341,19.578,153.419
C02445=1078.458,-106.897,-53.989,173.343,19.579,153.419
C02446=1078.464,-106.647,-53.999,173.345,19.580,153.419
C02447=1078.469,-106.398,-54.008,173.346,19.581,153.419
C02448=1078.476,-106.149,-54.019,173.348,19.583,153.419
C02449=1078.482,-105.899,-54.028,173.349,19.584,153.419
C02450=1078.488,-105.649,-54.038,173.351,19.585,153.419
C02451=1078.493,-105.399,-54.048,173.353,19.586,153.419
C02452=1078.500,-105.149,-54.058,173.354,19.587,153.419
C02453=1078.506,-104.900,-54.068,173.355,19.588,153.419
C02454=1078.512,-104.650,-54.077,173.357,19.589,153.419
C02455=1078.518,-104.400,-54.087,173.358,19.590,153.419
C02456=1078.525,-104.150,-54.097,173.360,19.591,153.419
C02457=1078.531,-103.900,-54.108,173.362,19.592,153.419
C02458=1078.537,-103.651,-54.117,173.363,19.594,153.419
C02459=1078.543,-103.401,-54.127,173.365,19.595,153.419
C02460=1078.549,-103.151,-54.137,173.367,19.596,153.418
C02461=1078.555,-102.902,-54.147,173.368,19.597,153.419
C02462=1078.561,-102.652,-54.157,173.370,19.598,153.418
C02463=1078.567,-102.402,-54.167,173.370,19.599,153.418
C02464=1078.573,-102.152,-54.177,173.372,19.600,153.418
C02465=1078.580,-101.903,-54.187,173.374,19.602,153.418
C02466=1078.586,-101.653,-54.196,173.375,19.603,153.418
C02467=1078.591,-101.403,-54.207,173.377,19.604,153.418
C02468=1078.598,-101.154,-54.217,173.378,19.605,153.418
C02469=1078.604,-100.904,-54.226,173.380,19.607,153.418
C02470=1078.610,-100.654,-54.237,173.382,19.608,153.418
C02471=1078.616,-100.404,-54.247,173.383,19.609,153.418
C02472=1078.622,-100.155,-54.256,173.385,19.610,153.418
C02473=1078.628,-99.905,-54.267,173.386,19.611,153.418
C02474=1078.634,-99.655,-54.277,173.387,19.612,153.418
C02475=1078.640,-99.406,-54.286,173.389,19.613,153.418
C02476=1078.647,-99.156,-54.297,173.390,19.614,153.418
C02477=1078.652,-98.906,-54.307,173.392,19.616,153.418
C02478=1078.659,-98.656,-54.318,173.394,19.617,153.418
C02479=1078.665,-98.407,-54.327,173.395,19.618,153.418
C02480=1078.671,-98.156,-54.337,173.397,19.619,153.418
C02481=1078.677,-97.877,-54.349,173.398,19.621,153.418
C02482=1078.685,-97.597,-54.361,173.400,19.622,153.418
C02483=1078.691,-97.317,-54.371,173.401,19.623,153.418
C02484=1078.698,-97.038,-54.383,173.404,19.625,153.418
C02485=1078.703,-96.789,-54.394,173.405,19.626,153.417
C02486=1078.710,-96.539,-54.403,173.406,19.627,153.418
C02487=1078.716,-96.288,-54.414,173.408,19.629,153.418
C02488=1078.722,-96.039,-54.424,173.409,19.630,153.417
C02489=1078.728,-95.789,-54.434,173.411,19.631,153.417
C02490=1078.734,-95.539,-54.444,173.412,19.633,153.417
C02491=1078.740,-95.289,-54.455,173.414,19.634,153.417
C02492=1078.746,-95.040,-54.465,173.415,19.635,153.417
C02493=1078.751,-94.790,-54.475,173.417,19.636,153.417
C02494=1078.758,-94.541,-54.485,173.419,19.637,153.417
C02495=1078.763,-94.291,-54.495,173.420,19.639,153.417
C02496=1078.770,-94.042,-54.506,173.422,19.640,153.417
C02497=1078.775,-93.791,-54.516,173.423,19.642,153.417
C02498=1078.782,-93.542,-54.526,173.425,19.643,153.417
C02499=1078.788,-93.291,-54.537,173.426,19.644,153.417
C02500=1078.794,-93.042,-54.547,173.428,19.646,153.417
C02501=1078.800,-92.793,-54.558,173.429,19.647,153.417
C02502=1078.806,-92.543,-54.567,173.431,19.648,153.417
C02503=1078.812,-92.294,-54.578,173.432,19.649,153.417
C02504=1078.817,-92.043,-54.588,173.433,19.651,153.417
C02505=1078.824,-91.794,-54.599,173.435,19.652,153.417
C02506=1078.829,-91.544,-54.609,173.436,19.653,153.417
C02507=1078.836,-91.294,-54.620,173.438,19.655,153.417
C02508=1078.842,-91.045,-54.630,173.439,19.656,153.417
C02509=1078.848,-90.795,-54.640,173.441,19.657,153.417
C02510=1078.854,-90.545,-54.651,173.442,19.659,153.417
C02511=1078.860,-90.296,-54.660,173.444,19.660,153.417
C02512=1078.866,-90.046,-54.671,173.445,19.662,153.417
C02513=1078.872,-89.796,-54.683,173.447,19.663,153.417
C02514=1078.878,-89.546,-54.692,173.449,19.664,153.417
C02515=1078.884,-89.297,-54.703,173.450,19.666,153.417
C02516=1078.891,-89.048,-54.713,173.452,19.667,153.417
C02517=1078.896,-88.797,-54.723,173.453,19.668,153.417
C02518=1078.902,-88.548,-54.734,173.455,19.669,153.417
C02519=1078.909,-88.298,-54.745,173.456,19.671,153.417
C02520=1078.914,-88.048,-54.755,173.458,19.672,153.417
C02521=1078.921,-87.799,-54.765,173.459,19.674,153.417
C02522=1078.926,-87.549,-54.776,173.461,19.675,153.417
C02523=1078.933,-87.298,-54.787,173.462,19.676,153.417
C02524=1078.939,-87.049,-54.797,173.464,19.678,153.417
C02525=1078.945,-86.800,-54.808,173.465,19.679,153.417
C02526=1078.951,-86.550,-54.818,173.467,19.681,153.417
C02527=1078.957,-86.301,-54.828,173.469,19.682,153.417
C02528=1078.963,-86.050,-54.840,173.469,19.683,153.417
C02529=1078.969,-85.801,-54.850,173.471,19.684,153.417
C02530=1078.975,-85.551,-54.860,173.472,19.686,153.417
C02531=1078.981,-85.302,-54.870,173.474,19.687,153.417
C02532=1078.988,-85.052,-54.882,173.475,19.689,153.417
C02533=1078.993,-84.802,-54.892,173.477,19.690,153.417
C02534=1079.000,-84.552,-54.902,173.478,19.691,153.417
C02535=1079.005,-84.303,-54.913,173.480,19.693,153.417
C02536=1079.012,-84.053,-54.924,173.481,19.694,153.417
C02537=1079.018,-83.804,-54.934,173.483,19.696,153.417
C02538=1079.024,-83.554,-54.945,173.484,19.697,153.417
C02539=1079.029,-83.304,-54.955,173.486,19.699,153.417
C02540=1079.036,-83.054,-54.966,173.487,19.700,153.417
C02541=1079.042,-82.805,-54.977,173.489,19.701,153.417
C02542=1079.048,-82.555,-54.988,173.490,19.703,153.417
C02543=1079.055,-82.305,-54.999,173.492,19.704,153.417
C02544=1079.061,-82.056,-55.009,173.493,19.706,153.417
C02545=1079.068,-81.778,-55.021,173.495,19.707,153.417
C02546=1079.074,-81.500,-55.032,173.497,19.709,153.417
C02547=1079.081,-81.223,-55.045,173.499,19.710,153.417
C02548=1079.088,-80.945,-55.056,173.500,19.712,153.417
C02549=1079.094,-80.696,-55.067,173.502,19.713,153.417
C02550=1079.100,-80.446,-55.078,173.503,19.715,153.417
C02551=1079.106,-80.196,-55.089,173.505,19.716,153.417
C02552=1079.113,-79.947,-55.099,173.506,19.718,153.417
C02553=1079.118,-79.697,-55.110,173.508,19.719,153.417
C02554=1079.125,-79.447,-55.121,173.509,19.721,153.417
C02555=1079.130,-79.198,-55.132,173.511,19.722,153.418
C02556=1079.136,-78.948,-55.143,173.512,19.724,153.418
C02557=1079.143,-78.699,-55.153,173.514,19.725,153.418
C02558=1079.149,-78.448,-55.164,173.515,19.727,153.418
C02559=1079.154,-78.199,-55.175,173.517,19.728,153.418
C02560=1079.160,-77.949,-55.186,173.518,19.730,153.418
C02561=1079.166,-77.699,-55.197,173.519,19.731,153.418
C02562=1079.172,-77.450,-55.208,173.521,19.733,153.418
C02563=1079.178,-77.200,-55.219,173.522,19.734,153.418
C02564=1079.185,-76.950,-55.229,173.524,19.736,153.418
C02565=1079.191,-76.701,-55.240,173.525,19.737,153.418
C02566=1079.197,-76.451,-55.251,173.527,19.739,153.418
C02567=1079.202,-76.202,-55.262,173.528,19.740,153.418
C02568=1079.209,-75.951,-55.273,173.530,19.742,153.418
C02569=1079.214,-75.702,-55.284,173.531,19.743,153.418
C02570=1079.220,-75.453,-55.295,173.533,19.745,153.418
C02571=1079.226,-75.202,-55.306,173.534,19.747,153.418
C02572=1079.232,-74.953,-55.317,173.536,19.748,153.418
C02573=1079.239,-74.703,-55.328,173.537,19.750,153.418
C02574=1079.245,-74.453,-55.339,173.539,19.751,153.418
C02575=1079.251,-74.204,-55.350,173.540,19.753,153.418
C02576=1079.257,-73.954,-55.361,173.542,19.754,153.418
C02577=1079.263,-73.704,-55.372,173.543,19.756,153.418
C02578=1079.269,-73.455,-55.383,173.544,19.757,153.418
C02579=1079.275,-73.206,-55.394,173.546,19.759,153.418
C02580=1079.280,-72.955,-55.406,173.547,19.761,153.418
C02581=1079.286,-72.706,-55.417,173.549,19.762,153.418
C02582=1079.292,-72.456,-55.428,173.550,19.764,153.418
C02583=1079.298,-72.206,-55.439,173.551,19.766,153.419
C02584=1079.304,-71.957,-55.450,173.553,19.767,153.419
C02585=1079.309,-71.707,-55.461,173.554,19.769,153.419
C02586=1079.316,-71.457,-55.472,173.557,19.770,153.419
C02587=1079.322,-71.208,-55.483,173.558,19.772,153.419
C02588=1079.328,-70.959,-55.494,173.559,19.774,153.419
C02589=1079.334,-70.709,-55.506,173.561,19.775,153.419
C02590=1079.339,-70.459,-55.517,173.562,19.777,153.419
C02591=1079.345,-70.209,-55.528,173.564,19.778,153.419
C02592=1079.351,-69.959,-55.539,173.565,19.780,153.419
C02593=1079.357,-69.710,-55.550,173.567,19.782,153.419
C02594=1079.363,-69.461,-55.562,173.568,19.783,153.419
C02595=1079.369,-69.211,-55.573,173.570,19.785,153.419
C02596=1079.375,-68.961,-55.584,173.571,19.787,153.419
C02597=1079.381,-68.711,-55.595,173.572,19.788,153.419
C02598=1079.386,-68.461,-55.607,173.574,19.790,153.419
C02599=1079.392,-68.212,-55.617,173.575,19.792,153.420
C02600=1079.399,-67.962,-55.629,173.577,19.793,153.420
C02601=1079.404,-67.712,-55.640,173.578,19.795,153.420
C02602=1079.410,-67.463,-55.651,173.580,19.796,153.420
C02603=1079.416,-67.213,-55.662,173.581,19.798,153.420
C02604=1079.422,-66.964,-55.674,173.582,19.800,153.420
C02605=1079.428,-66.713,-55.686,173.584,19.801,153.420
C02606=1079.434,-66.464,-55.697,173.585,19.803,153.420
C02607=1079.440,-66.214,-55.708,173.587,19.805,153.420
C02608=1079.446,-65.965,-55.720,173.588,19.806,153.420
C02609=1079.452,-65.690,-55.732,173.590,19.809,153.420
C02610=1079.459,-65.414,-55.744,173.592,19.810,153.420
C02611=1079.465,-65.139,-55.757,173.593,19.812,153.420
C02612=1079.473,-64.864,-55.770,173.595,19.814,153.420
C02613=1079.478,-64.614,-55.781,173.597,19.816,153.420
C02614=1079.484,-64.364,-55.792,173.598,19.818,153.421
C02615=1079.490,-64.114,-55.803,173.599,19.819,153.421
C02616=1079.496,-63.865,-55.815,173.601,19.821,153.421
C02617=1079.502,-63.615,-55.826,173.602,19.823,153.421
C02618=1079.509,-63.366,-55.838,173.604,19.824,153.421
C02619=1079.514,-63.116,-55.849,173.605,19.826,153.421
C02620=1079.520,-62.866,-55.861,173.606,19.828,153.421
C02621=1079.526,-62.617,-55.872,173.608,19.829,153.421
C02622=1079.532,-62.366,-55.884,173.609,19.831,153.421
C02623=1079.538,-62.117,-55.895,173.611,19.833,153.421
C02624=1079.544,-61.867,-55.907,173.612,19.834,153.421
C02625=1079.550,-61.618,-55.918,173.614,19.836,153.421
C02626=1079.556,-61.368,-55.930,173.615,19.838,153.422
C02627=1079.562,-61.119,-55.941,173.616,19.839,153.422
C02628=1079.569,-60.868,-55.952,173.619,19.841,153.422
C02629=1079.574,-60.619,-55.964,173.620,19.843,153.422
C02630=1079.580,-60.369,-55.975,173.621,19.845,153.422
C02631=1079.586,-60.120,-55.987,173.623,19.847,153.422
C02632=1079.593,-59.870,-55.998,173.624,19.848,153.422
C02633=1079.598,-59.621,-56.011,173.626,19.850,153.422
C02634=1079.604,-59.371,-56.022,173.627,19.852,153.422
C02635=1079.610,-59.121,-56.033,173.628,19.853,153.422
C02636=1079.617,-58.871,-56.045,173.630,19.855,153.422
C02637=1079.622,-58.622,-56.056,173.631,19.857,153.422
C02638=1079.628,-58.372,-56.068,173.633,19.858,153.422
C02639=1079.634,-58.123,-56.079,173.634,19.860,153.423
C02640=1079.641,-57.873,-56.091,173.635,19.862,153.423
C02641=1079.646,-57.623,-56.103,173.637,19.863,153.423
C02642=1079.652,-57.374,-56.114,173.639,19.866,153.423
C02643=1079.659,-57.123,-56.126,173.641,19.867,153.423
C02644=1079.665,-56.875,-56.137,173.642,19.869,153.423
C02645=1079.670,-56.624,-56.149,173.643,19.871,153.423
C02646=1079.676,-56.375,-56.161,173.645,19.872,153.423
C02647=1079.683,-56.126,-56.173,173.646,19.874,153.423
C02648=1079.689,-55.875,-56.184,173.647,19.876,153.423
C02649=1079.695,-55.626,-56.196,173.649,19.878,153.423
C02650=1079.701,-55.376,-56.207,173.650,19.879,153.423
C02651=1079.707,-55.127,-56.219,173.652,19.881,153.424
C02652=1079.713,-54.877,-56.231,173.653,19.883,153.424
C02653=1079.719,-54.627,-56.243,173.654,19.884,153.424
C02654=1079.725,-54.378,-56.254,173.657,19.886,153.424
C02655=1079.731,-54.128,-56.266,173.658,19.888,153.424
C02656=1079.738,-53.878,-56.278,173.659,19.890,153.424
C02657=1079.743,-53.629,-56.289,173.661,19.891,153.424
C02658=1079.749,-53.379,-56.301,173.662,19.893,153.424
C02659=1079.755,-53.130,-56.313,173.664,19.895,153.424
C02660=1079.762,-52.880,-56.324,173.665,19.897,153.424
C02661=1079.768,-52.630,-56.336,173.666,19.898,153.424
C02662=1079.774,-52.381,-56.348,173.668,19.900,153.424
C02663=1079.780,-52.131,-56.360,173.669,19.902,153.424
C02664=1079.787,-51.881,-56.372,173.671,19.903,153.425
C02665=1079.792,-51.632,-56.384,173.673,19.906,153.425
C02666=1079.798,-51.382,-56.395,173.674,19.907,153.425
C02667=1079.805,-51.132,-56.407,173.675,19.909,153.425
C02668=1079.810,-50.883,-56.419,173.677,19.911,153.425
C02669=1079.816,-50.633,-56.430,173.678,19.913,153.425
C02670=1079.822,-50.383,-56.443,173.680,19.914,153.425
C02671=1079.828,-50.134,-56.455,173.681,19.916,153.425
C02672=1079.834,-49.884,-56.467,173.682,19.918,153.425
C02673=1079.841,-49.610,-56.480,173.685,19.920,153.425
C02674=1079.847,-49.335,-56.493,173.686,19.922,153.426
C02675=1079.854,-49.062,-56.506,173.687,19.924,153.426
C02676=1079.860,-48.788,-56.519,173.688,19.926,153.426
C02677=1079.866,-48.538,-56.532,173.691,19.928,153.426
C02678=1079.872,-48.289,-56.543,173.692,19.930,153.426
C02679=1079.878,-48.039,-56.556,173.693,19.932,153.426
C02680=1079.884,-47.790,-56.567,173.695,19.934,153.426
C02681=1079.890,-47.540,-56.579,173.696,19.936,153.426
C02682=1079.896,-47.290,-56.592,173.697,19.937,153.426
C02683=1079.902,-47.041,-56.603,173.699,19.939,153.427
C02684=1079.908,-46.791,-56.616,173.700,19.941,153.427
C02685=1079.914,-46.541,-56.627,173.701,19.943,153.427
C02686=1079.919,-46.292,-56.639,173.704,19.945,153.427
C02687=1079.925,-46.042,-56.652,173.705,19.947,153.427
C02688=1079.932,-45.792,-56.664,173.706,19.949,153.427
C02689=1079.937,-45.543,-56.676,173.708,19.951,153.427
C02690=1079.944,-45.294,-56.688,173.709,19.952,153.427
C02691=1079.950,-45.044,-56.700,173.710,19.954,153.427
C02692=1079.955,-44.794,-56.712,173.712,19.956,153.428
C02693=1079.961,-44.544,-56.724,173.713,19.958,153.428
C02694=1079.967,-44.294,-56.736,173.715,19.960,153.428
C02695=1079.973,-44.044,-56.749,173.716,19.962,153.428
C02696=1079.979,-43.796,-56.761,173.718,19.964,153.428
C02697=1079.985,-43.546,-56.773,173.719,19.966,153.428
C02698=1079.991,-43.296,-56.786,173.720,19.968,153.428
C02699=1079.997,-43.047,-56.797,173.722,19.969,153.428
C02700=1080.003,-42.797,-56.810,173.723,19.971,153.429
C02701=1080.009,-42.547,-56.822,173.725,19.973,153.429
C02702=1080.015,-42.297,-56.834,173.727,19.975,153.429
C02703=1080.020,-42.048,-56.846,173.728,19.977,153.429
C02704=1080.026,-41.798,-56.858,173.729,19.979,153.429
C02705=1080.033,-41.548,-56.870,173.731,19.981,153.429
C02706=1080.039,-41.298,-56.883,173.732,19.983,153.429
C02707=1080.044,-41.049,-56.895,173.733,19.985,153.429
C02708=1080.051,-40.800,-56.907,173.735,19.987,153.430
C02709=1080.057,-40.550,-56.920,173.736,19.988,153.430
C02710=1080.063,-40.300,-56.932,173.738,19.991,153.430
C02711=1080.069,-40.051,-56.944,173.740,19.993,153.430
C02712=1080.075,-39.801,-56.956,173.741,19.994,153.430
C02713=1080.081,-39.551,-56.969,173.742,19.996,153.430
C02714=1080.086,-39.301,-56.981,173.744,19.998,153.430
C02715=1080.093,-39.053,-56.993,173.745,20.000,153.430
C02716=1080.098,-38.803,-57.006,173.746,20.002,153.430
C02717=1080.104,-38.553,-57.018,173.748,20.004,153.431
C02718=1080.110,-38.303,-57.031,173.750,20.006,153.431
C02719=1080.116,-38.054,-57.042,173.751,20.008,153.431
C02720=1080.122,-37.804,-57.055,173.752,20.010,153.431
C02721=1080.128,-37.555,-57.068,173.754,20.012,153.431
C02722=1080.134,-37.305,-57.081,173.755,20.014,153.431
C02723=1080.140,-37.056,-57.093,173.756,20.016,153.431
C02724=1080.146,-36.806,-57.105,173.758,20.017,153.431
C02725=1080.151,-36.556,-57.118,173.760,20.020,153.432
C02726=1080.157,-36.306,-57.131,173.761,20.022,153.432
C02727=1080.164,-36.057,-57.142,173.762,20.024,153.432
C02728=1080.169,-35.807,-57.155,173.764,20.026,153.432
C02729=1080.175,-35.558,-57.167,173.765,20.027,153.432
C02730=1080.181,-35.308,-57.180,173.766,20.029,153.432
C02731=1080.187,-35.058,-57.193,173.768,20.031,153.432
C02732=1080.193,-34.809,-57.205,173.770,20.034,153.433
C02733=1080.199,-34.559,-57.218,173.771,20.036,153.433
C02734=1080.204,-34.309,-57.230,173.772,20.038,153.433
C02735=1080.210,-34.060,-57.243,173.774,20.039,153.433
C02736=1080.216,-33.810,-57.255,173.775,20.041,153.433
C02737=1080.223,-33.537,-57.269,173.777,20.044,153.433
C02738=1080.230,-33.263,-57.283,173.779,20.046,153.433
C02739=1080.236,-32.989,-57.297,173.780,20.048,153.434
C02740=1080.243,-32.715,-57.311,173.782,20.050,153.434
C02741=1080.248,-32.466,-57.323,173.783,20.052,153.434
C02742=1080.254,-32.217,-57.336,173.784,20.054,153.434
C02743=1080.260,-31.967,-57.349,173.786,20.056,153.434
C02744=1080.266,-31.717,-57.361,173.787,20.058,153.434
C02745=1080.272,-31.467,-57.374,173.788,20.060,153.434
C02746=1080.278,-31.218,-57.387,173.791,20.062,153.435
C02747=1080.285,-30.968,-57.399,173.792,20.064,153.435
C02748=1080.290,-30.719,-57.411,173.793,20.066,153.435
C02749=1080.296,-30.469,-57.424,173.794,20.068,153.435
C02750=1080.302,-30.220,-57.437,173.796,20.070,153.435
C02751=1080.308,-29.970,-57.450,173.797,20.072,153.435
C02752=1080.314,-29.720,-57.462,173.799,20.074,153.435
C02753=1080.320,-29.471,-57.476,173.801,20.076,153.436
C02754=1080.326,-29.221,-57.488,173.802,20.078,153.436
C02755=1080.332,-28.971,-57.501,173.803,20.080,153.436
C02756=1080.337,-28.722,-57.513,173.804,20.082,153.436
C02757=1080.344,-28.473,-57.526,173.806,20.084,153.436
C02758=1080.349,-28.223,-57.539,173.808,20.086,153.436
C02759=1080.356,-27.974,-57.552,173.809,20.088,153.436
C02760=1080.362,-27.724,-57.564,173.811,20.090,153.437
C02761=1080.367,-27.474,-57.577,173.812,20.092,153.437
C02762=1080.374,-27.225,-57.590,173.813,20.094,153.437
C02763=1080.380,-26.975,-57.603,173.814,20.096,153.437
C02764=1080.385,-26.725,-57.615,173.816,20.099,153.437
C02765=1080.392,-26.476,-57.629,173.818,20.100,153.437
C02766=1080.398,-26.226,-57.641,173.819,20.102,153.437
C02767=1080.402,-25.977,-57.655,173.820,20.104,153.438
C02768=1080.408,-25.727,-57.667,173.822,20.106,153.438
C02769=1080.414,-25.477,-57.680,173.823,20.108,153.438
C02770=1080.421,-25.228,-57.693,173.825,20.110,153.438
C02771=1080.426,-24.978,-57.706,173.826,20.112,153.438
C02772=1080.433,-24.729,-57.719,173.828,20.114,153.438
C02773=1080.438,-24.478,-57.732,173.829,20.116,153.439
C02774=1080.444,-24.229,-57.745,173.830,20.118,153.439
C02775=1080.450,-23.979,-57.758,173.832,20.120,153.439
C02776=1080.456,-23.730,-57.771,173.834,20.123,153.439
C02777=1080.462,-23.480,-57.784,173.835,20.125,153.439
C02778=1080.467,-23.231,-57.796,173.836,20.127,153.439
C02779=1080.473,-22.981,-57.810,173.837,20.129,153.440
C02780=1080.479,-22.732,-57.822,173.839,20.131,153.440
C02781=1080.485,-22.482,-57.836,173.840,20.133,153.440
C02782=1080.491,-22.232,-57.848,173.842,20.135,153.440
C02783=1080.496,-21.983,-57.862,173.843,20.137,153.440
C02784=1080.503,-21.734,-57.875,173.845,20.139,153.440
C02785=1080.508,-21.484,-57.888,173.846,20.141,153.440
C02786=1080.515,-21.234,-57.901,173.847,20.143,153.441
C02787=1080.521,-20.985,-57.914,173.849,20.146,153.441
C02788=1080.526,-20.735,-57.928,173.851,20.148,153.441
C02789=1080.532,-20.485,-57.940,173.852,20.150,153.441
C02790=1080.538,-20.236,-57.953,173.853,20.151,153.441
C02791=1080.544,-19.986,-57.966,173.855,20.153,153.441
C02792=1080.550,-19.736,-57.980,173.857,20.156,153.441
C02793=1080.556,-19.487,-57.993,173.858,20.158,153.442
C02794=1080.562,-19.237,-58.006,173.859,20.160,153.442
C02795=1080.568,-18.988,-58.019,173.861,20.162,153.442
C02796=1080.573,-18.738,-58.032,173.862,20.164,153.442
C02797=1080.579,-18.488,-58.045,173.863,20.166,153.442
C02798=1080.585,-18.239,-58.059,173.865,20.168,153.442
C02799=1080.591,-17.989,-58.071,173.867,20.170,153.443
C02800=1080.597,-17.740,-58.085,173.868,20.172,153.443
C02801=1080.604,-17.465,-58.099,173.869,20.174,153.443
C02802=1080.610,-17.191,-58.114,173.871,20.177,153.443
C02803=1080.617,-16.917,-58.129,173.872,20.179,153.443
C02804=1080.623,-16.642,-58.143,173.874,20.182,153.443
C02805=1080.629,-16.392,-58.156,173.876,20.184,153.444
C02806=1080.636,-16.142,-58.169,173.877,20.186,153.444
C02807=1080.642,-15.893,-58.183,173.878,20.188,153.444
C02808=1080.647,-15.644,-58.197,173.880,20.190,153.444
C02809=1080.653,-15.394,-58.209,173.882,20.192,153.444
C02810=1080.659,-15.144,-58.222,173.883,20.194,153.444
C02811=1080.665,-14.895,-58.236,173.884,20.196,153.445
C02812=1080.671,-14.645,-58.249,173.885,20.198,153.445
C02813=1080.676,-14.395,-58.263,173.887,20.200,153.445
C02814=1080.682,-14.146,-58.276,173.889,20.203,153.445
C02815=1080.689,-13.897,-58.289,173.890,20.205,153.445
C02816=1080.694,-13.647,-58.302,173.891,20.207,153.445
C02817=1080.700,-13.397,-58.316,173.893,20.209,153.446
C02818=1080.705,-13.148,-58.329,173.894,20.211,153.446
C02819=1080.712,-12.899,-58.343,173.896,20.213,153.446
C02820=1080.717,-12.649,-58.357,173.897,20.215,153.446
C02821=1080.723,-12.399,-58.369,173.898,20.218,153.446
C02822=1080.729,-12.150,-58.383,173.900,20.220,153.447
C02823=1080.735,-11.900,-58.396,173.901,20.222,153.447
C02824=1080.740,-11.651,-58.410,173.903,20.224,153.447
C02825=1080.747,-11.401,-58.424,173.904,20.226,153.447
C02826=1080.753,-11.151,-58.438,173.906,20.228,153.447
C02827=1080.758,-10.901,-58.450,173.907,20.230,153.447
C02828=1080.764,-10.652,-58.464,173.908,20.232,153.448
C02829=1080.770,-10.402,-58.477,173.910,20.235,153.448
C02830=1080.776,-10.153,-58.491,173.912,20.237,153.448
C02831=1080.782,-9.904,-58.504,173.913,20.239,153.448
C02832=1080.787,-9.654,-58.518,173.914,20.241,153.448
C02833=1080.794,-9.405,-58.532,173.915,20.243,153.448
C02834=1080.799,-9.155,-58.545,173.917,20.246,153.449
C02835=1080.805,-8.905,-58.558,173.919,20.248,153.449
C02836=1080.811,-8.655,-58.572,173.920,20.250,153.449
C02837=1080.817,-8.406,-58.586,173.921,20.252,153.449
C02838=1080.823,-8.156,-58.599,173.923,20.254,153.449
C02839=1080.829,-7.907,-58.613,173.925,20.256,153.449
C02840=1080.834,-7.657,-58.627,173.926,20.258,153.450
C02841=1080.841,-7.408,-58.640,173.927,20.260,153.450
C02842=1080.847,-7.158,-58.654,173.928,20.262,153.450
C02843=1080.853,-6.909,-58.667,173.931,20.264,153.450
C02844=1080.858,-6.659,-58.681,173.932,20.266,153.450
C02845=1080.864,-6.409,-58.695,173.933,20.268,153.450
C02846=1080.870,-6.160,-58.708,173.934,20.270,153.451
C02847=1080.875,-5.911,-58.722,173.936,20.272,153.451
C02848=1080.882,-5.661,-58.736,173.938,20.275,153.451
C02849=1080.888,-5.411,-58.750,173.939,20.277,153.451
C02850=1080.894,-5.162,-58.763,173.940,20.279,153.451
C02851=1080.899,-4.912,-58.777,173.941,20.281,153.452
C02852=1080.906,-4.663,-58.790,173.944,20.284,153.452
C02853=1080.911,-4.413,-58.804,173.945,20.286,153.452
C02854=1080.917,-4.163,-58.818,173.946,20.288,153.452
C02855=1080.923,-3.914,-58.831,173.947,20.290,153.452
C02856=1080.929,-3.664,-58.845,173.949,20.292,153.452
C02857=1080.935,-3.415,-58.859,173.951,20.294,153.452
C02858=1080.941,-3.165,-58.873,173.952,20.296,153.453
C02859=1080.947,-2.915,-58.887,173.953,20.298,153.453
C02860=1080.952,-2.666,-58.901,173.954,20.301,153.453
C02861=1080.959,-2.417,-58.914,173.957,20.303,153.453
C02862=1080.964,-2.167,-58.928,173.958,20.305,153.453
C02863=1080.970,-1.918,-58.942,173.959,20.307,153.454
C02864=1080.975,-1.668,-58.956,173.960,20.309,153.454
C02865=1080.982,-1.392,-58.971,173.962,20.312,153.454
C02866=1080.988,-1.116,-58.986,173.964,20.314,153.454
C02867=1080.994,-0.840,-59.002,173.966,20.317,153.454
C02868=1081.001,-0.564,-59.017,173.967,20.319,153.455
C02869=1081.007,-0.314,-59.032,173.968,20.321,153.455
C02870=1081.013,-0.064,-59.046,173.970,20.324,153.455
C02871=1081.018,0.185,-59.059,173.971,20.326,153.455
C02872=1081.024,0.434,-59.074,173.973,20.328,153.455
C02873=1081.030,0.684,-59.087,173.974,20.330,153.456
C02874=1081.036,0.934,-59.101,173.976,20.333,153.456
C02875=1081.042,1.184,-59.115,173.977,20.335,153.456
C02876=1081.047,1.433,-59.129,173.978,20.337,153.456
C02877=1081.053,1.682,-59.144,173.980,20.339,153.456
C02878=1081.058,1.932,-59.158,173.981,20.341,153.457
C02879=1081.065,2.182,-59.171,173.983,20.344,153.457
C02880=1081.071,2.431,-59.185,173.984,20.346,153.457
C02881=1081.076,2.680,-59.200,173.986,20.348,153.457
C02882=1081.082,2.930,-59.214,173.987,20.350,153.457
C02883=1081.088,3.180,-59.228,173.989,20.353,153.457
C02884=1081.093,3.430,-59.242,173.990,20.355,153.458
C02885=1081.099,3.679,-59.256,173.991,20.357,153.458
C02886=1081.105,3.928,-59.270,173.993,20.359,153.458
C02887=1081.112,4.178,-59.284,173.995,20.362,153.458
C02888=1081.117,4.427,-59.298,173.996,20.364,153.458
C02889=1081.123,4.677,-59.312,173.997,20.366,153.459
C02890=1081.128,4.926,-59.326,173.998,20.368,153.459
C02891=1081.135,5.176,-59.341,174.001,20.370,153.459
C02892=1081.140,5.425,-59.355,174.002,20.372,153.459
C02893=1081.146,5.675,-59.369,174.003,20.374,153.459
C02894=1081.152,5.925,-59.384,174.004,20.376,153.460
C02895=1081.158,6.174,-59.397,174.006,20.379,153.460
C02896=1081.164,6.423,-59.411,174.008,20.381,153.460
C02897=1081.170,6.673,-59.426,174.009,20.383,153.460
C02898=1081.176,6.923,-59.440,174.010,20.385,153.460
C02899=1081.181,7.172,-59.454,174.012,20.388,153.460
C02900=1081.187,7.422,-59.468,174.013,20.390,153.461
C02901=1081.193,7.672,-59.482,174.015,20.392,153.461
C02902=1081.199,7.920,-59.497,174.016,20.394,153.461
C02903=1081.205,8.171,-59.511,174.018,20.396,153.461
C02904=1081.211,8.420,-59.526,174.019,20.398,153.461
C02905=1081.216,8.669,-59.540,174.021,20.400,153.461
C02906=1081.223,8.919,-59.553,174.022,20.403,153.462
C02907=1081.229,9.168,-59.568,174.024,20.405,153.462
C02908=1081.234,9.418,-59.582,174.025,20.407,153.462
C02909=1081.240,9.667,-59.597,174.027,20.409,153.462
C02910=1081.246,9.917,-59.610,174.028,20.411,153.462
C02911=1081.252,10.166,-59.625,174.030,20.414,153.463
C02912=1081.258,10.416,-59.639,174.031,20.416,153.463
C02913=1081.264,10.665,-59.654,174.032,20.418,153.463
C02914=1081.270,10.915,-59.668,174.034,20.420,153.463
C02915=1081.275,11.164,-59.683,174.036,20.423,153.463
C02916=1081.281,11.414,-59.697,174.037,20.425,153.463
C02917=1081.287,11.664,-59.711,174.038,20.427,153.464
C02918=1081.293,11.913,-59.725,174.040,20.429,153.464
C02919=1081.299,12.163,-59.740,174.042,20.432,153.464
C02920=1081.305,12.412,-59.755,174.043,20.434,153.464
C02921=1081.311,12.662,-59.769,174.044,20.436,153.464
C02922=1081.317,12.911,-59.784,174.045,20.438,153.465
C02923=1081.322,13.161,-59.798,174.048,20.440,153.465
C02924=1081.329,13.410,-59.813,174.049,20.442,153.465
C02925=1081.334,13.660,-59.826,174.050,20.444,153.465
C02926=1081.341,13.910,-59.841,174.051,20.446,153.465
C02927=1081.346,14.159,-59.856,174.053,20.449,153.466
C02928=1081.352,14.409,-59.870,174.055,20.451,153.466
C02929=1081.359,14.686,-59.886,174.056,20.453,153.466
C02930=1081.365,14.965,-59.902,174.058,20.456,153.466
C02931=1081.372,15.242,-59.919,174.059,20.458,153.466
C02932=1081.378,15.521,-59.936,174.061,20.461,153.467
C02933=1081.384,15.770,-59.949,174.062,20.463,153.467
C02934=1081.389,16.019,-59.964,174.065,20.465,153.467
C02935=1081.396,16.269,-59.979,174.066,20.467,153.467
C02936=1081.401,16.519,-59.993,174.067,20.469,153.467
C02937=1081.408,16.768,-60.008,174.068,20.472,153.468
C02938=1081.413,17.018,-60.023,174.070,20.474,153.468
C02939=1081.419,17.268,-60.037,174.072,20.476,153.468
C02940=1081.425,17.517,-60.052,174.073,20.478,153.468
C02941=1081.430,17.766,-60.066,174.074,20.480,153.468
C02942=1081.437,18.015,-60.081,174.076,20.483,153.468
C02943=1081.442,18.265,-60.096,174.077,20.485,153.469
C02944=1081.448,18.515,-60.111,174.079,20.487,153.469
C02945=1081.454,18.764,-60.125,174.080,20.489,153.469
C02946=1081.460,19.014,-60.140,174.082,20.492,153.469
C02947=1081.466,19.263,-60.154,174.083,20.494,153.469
C02948=1081.471,19.513,-60.170,174.085,20.496,153.470
C02949=1081.477,19.762,-60.184,174.087,20.498,153.470
C02950=1081.483,20.012,-60.199,174.088,20.500,153.470
C02951=1081.489,20.261,-60.213,174.089,20.502,153.470
C02952=1081.494,20.511,-60.229,174.090,20.505,153.470
C02953=1081.500,20.760,-60.243,174.092,20.507,153.470
C02954=1081.507,21.010,-60.258,174.094,20.509,153.471
C02955=1081.512,21.259,-60.273,174.095,20.511,153.471
C02956=1081.517,21.508,-60.288,174.097,20.514,153.471
C02957=1081.524,21.758,-60.302,174.098,20.516,153.471
C02958=1081.529,22.007,-60.317,174.100,20.518,153.471
C02959=1081.535,22.257,-60.332,174.101,20.520,153.472
C02960=1081.541,22.506,-60.347,174.103,20.523,153.472
C02961=1081.547,22.756,-60.362,174.104,20.525,153.472
C02962=1081.552,23.005,-60.377,174.105,20.527,153.472
C02963=1081.559,23.255,-60.392,174.107,20.529,153.472
C02964=1081.564,23.504,-60.406,174.109,20.532,153.473
C02965=1081.570,23.754,-60.421,174.110,20.534,153.473
C02966=1081.576,24.004,-60.436,174.111,20.536,153.473
C02967=1081.581,24.253,-60.451,174.113,20.539,153.473
C02968=1081.587,24.503,-60.466,174.115,20.541,153.473
C02969=1081.593,24.752,-60.481,174.116,20.543,153.474
C02970=1081.599,25.002,-60.496,174.118,20.545,153.474
C02971=1081.605,25.251,-60.511,174.119,20.547,153.474
C02972=1081.611,25.500,-60.526,174.120,20.549,153.474
C02973=1081.616,25.750,-60.541,174.122,20.551,153.474
C02974=1081.622,25.999,-60.556,174.124,20.554,153.474
C02975=1081.628,26.248,-60.571,174.125,20.556,153.475
C02976=1081.634,26.498,-60.586,174.126,20.558,153.475
C02977=1081.640,26.748,-60.601,174.128,20.561,153.475
C02978=1081.645,26.997,-60.616,174.130,20.563,153.475
C02979=1081.652,27.247,-60.631,174.131,20.565,153.475
C02980=1081.657,27.496,-60.646,174.132,20.567,153.476
C02981=1081.663,27.746,-60.661,174.134,20.569,153.476
C02982=1081.669,27.995,-60.676,174.136,20.572,153.476
C02983=1081.675,28.245,-60.692,174.137,20.574,153.476
C02984=1081.681,28.494,-60.706,174.139,20.576,153.476
C02985=1081.686,28.744,-60.722,174.140,20.578,153.476
C02986=1081.692,28.993,-60.737,174.142,20.580,153.477
C02987=1081.697,29.243,-60.752,174.143,20.583,153.477
C02988=1081.704,29.492,-60.767,174.145,20.585,153.477
C02989=1081.709,29.742,-60.782,174.146,20.587,153.477
C02990=1081.715,29.991,-60.797,174.147,20.589,153.477
C02991=1081.721,30.241,-60.813,174.149,20.592,153.478
C02992=1081.726,30.490,-60.828,174.151,20.594,153.478
C02993=1081.733,30.769,-60.845,174.153,20.596,153.478
C02994=1081.739,31.049,-60.862,174.154,20.599,153.478
C02995=1081.746,31.328,-60.879,174.156,20.601,153.478
C02996=1081.752,31.608,-60.896,174.157,20.604,153.479
C02997=1081.758,31.858,-60.912,174.159,20.606,153.479
C02998=1081.764,32.107,-60.926,174.161,20.608,153.479
C02999=1081.770,32.356,-60.942,174.162,20.610,153.479
C03000=1081.776,32.606,-60.957,174.164,20.613,153.480
C03001=1081.782,32.856,-60.973,174.165,20.615,153.480
C03002=1081.787,33.105,-60.988,174.166,20.617,153.480
C03003=1081.793,33.354,-61.003,174.168,20.619,153.480
C03004=1081.798,33.603,-61.019,174.170,20.622,153.480
C03005=1081.805,33.853,-61.034,174.171,20.624,153.480
C03006=1081.810,34.103,-61.049,174.172,20.626,153.481
C03007=1081.815,34.352,-61.065,174.174,20.628,153.481
C03008=1081.822,34.602,-61.079,174.176,20.630,153.481
C03009=1081.828,34.851,-61.096,174.177,20.632,153.481
C03010=1081.834,35.100,-61.110,174.179,20.635,153.481
C03011=1081.839,35.350,-61.126,174.180,20.637,153.482
C03012=1081.845,35.599,-61.142,174.182,20.639,153.482
C03013=1081.851,35.848,-61.157,174.184,20.642,153.482
C03014=1081.857,36.098,-61.172,174.185,20.644,153.482
C03015=1081.862,36.348,-61.188,174.186,20.646,153.482
C03016=1081.869,36.597,-61.203,174.188,20.649,153.483
C03017=1081.874,36.846,-61.219,174.190,20.651,153.483
C03018=1081.880,37.096,-61.234,174.191,20.653,153.483
C03019=1081.886,37.345,-61.250,174.193,20.655,153.483
C03020=1081.891,37.595,-61.265,174.194,20.657,153.483
C03021=1081.898,37.844,-61.280,174.196,20.659,153.483
C03022=1081.904,38.094,-61.296,174.198,20.662,153.484
C03023=1081.909,38.344,-61.312,174.199,20.664,153.484
C03024=1081.914,38.593,-61.327,174.200,20.666,153.484
C03025=1081.920,38.842,-61.343,174.201,20.668,153.484
C03026=1081.927,39.092,-61.358,174.203,20.671,153.484
C03027=1081.932,39.341,-61.374,174.205,20.673,153.485
C03028=1081.938,39.591,-61.390,174.206,20.675,153.485
C03029=1081.943,39.841,-61.405,174.208,20.677,153.485
C03030=1081.949,40.089,-61.421,174.209,20.679,153.485
C03031=1081.955,40.339,-61.436,174.211,20.682,153.485
C03032=1081.961,40.588,-61.452,174.213,20.684,153.485
C03033=1081.966,40.837,-61.467,174.214,20.686,153.486
C03034=1081.972,41.087,-61.484,174.215,20.688,153.486
C03035=1081.978,41.337,-61.499,174.218,20.691,153.486
C03036=1081.983,41.587,-61.515,174.219,20.693,153.486
C03037=1081.989,41.835,-61.530,174.220,20.695,153.486
C03038=1081.995,42.085,-61.545,174.222,20.697,153.487
C03039=1082.001,42.334,-61.562,174.223,20.699,153.487
C03040=1082.007,42.584,-61.577,174.225,20.701,153.487
C03041=1082.012,42.833,-61.593,174.227,20.704,153.487
C03042=1082.018,43.083,-61.609,174.228,20.706,153.487
C03043=1082.024,43.332,-61.624,174.229,20.708,153.488
C03044=1082.030,43.581,-61.641,174.231,20.711,153.488
C03045=1082.036,43.831,-61.656,174.233,20.713,153.488
C03046=1082.041,44.080,-61.672,174.235,20.715,153.488
C03047=1082.047,44.330,-61.688,174.236,20.718,153.488
C03048=1082.053,44.579,-61.704,174.237,20.720,153.488
C03049=1082.058,44.829,-61.719,174.239,20.722,153.489
C03050=1082.064,45.078,-61.735,174.241,20.724,153.489
C03051=1082.070,45.328,-61.751,174.242,20.727,153.489
C03052=1082.075,45.577,-61.767,174.244,20.729,153.489
C03053=1082.081,45.826,-61.783,174.245,20.731,153.489
C03054=1082.086,46.076,-61.799,174.247,20.733,153.490
C03055=1082.092,46.325,-61.815,174.249,20.736,153.490
C03056=1082.097,46.575,-61.831,174.250,20.738,153.490
C03057=1082.104,46.854,-61.849,174.252,20.740,153.490
C03058=1082.110,47.134,-61.866,174.253,20.743,153.490
C03059=1082.117,47.413,-61.885,174.255,20.745,153.491
C03060=1082.123,47.693,-61.902,174.257,20.748,153.491
C03061=1082.129,47.942,-61.919,174.259,20.750,153.491
C03062=1082.134,48.191,-61.934,174.260,20.752,153.491
C03063=1082.140,48.441,-61.951,174.262,20.755,153.491
C03064=1082.146,48.690,-61.967,174.263,20.757,153.492
C03065=1082.151,48.940,-61.982,174.264,20.759,153.492
C03066=1082.157,49.190,-61.999,174.267,20.761,153.492
C03067=1082.162,49.438,-62.015,174.268,20.763,153.492
C03068=1082.168,49.688,-62.030,174.269,20.765,153.492
C03069=1082.174,49.938,-62.046,174.271,20.768,153.493
C03070=1082.180,50.187,-62.063,174.272,20.770,153.493
C03071=1082.186,50.436,-62.079,174.274,20.772,153.493
C03072=1082.192,50.686,-62.094,174.276,20.775,153.493
C03073=1082.197,50.935,-62.110,174.277,20.777,153.493
C03074=1082.202,51.185,-62.127,174.279,20.779,153.493
C03075=1082.208,51.434,-62.143,174.280,20.782,153.494
C03076=1082.214,51.683,-62.160,174.282,20.784,153.494
C03077=1082.220,51.933,-62.175,174.284,20.786,153.494
C03078=1082.226,52.183,-62.191,174.285,20.788,153.494
C03079=1082.232,52.432,-62.208,174.287,20.790,153.494
C03080=1082.237,52.681,-62.224,174.289,20.792,153.494
C03081=1082.244,52.982,-62.243,174.291,20.795,153.495
C03082=1082.251,53.284,-62.263,174.292,20.798,153.495
C03083=1082.258,53.585,-62.282,174.294,20.800,153.495
C03084=1082.265,53.887,-62.302,174.296,20.803,153.495
C03085=1082.271,54.136,-62.318,174.297,20.805,153.496
C03086=1082.276,54.386,-62.334,174.299,20.808,153.496
C03087=1082.282,54.635,-62.350,174.301,20.810,153.496
C03088=1082.288,54.885,-62.367,174.303,20.812,153.496
C03089=1082.294,55.134,-62.383,174.304,20.814,153.496
C03090=1082.299,55.384,-62.400,174.305,20.816,153.496
C03091=1082.305,55.632,-62.416,174.307,20.819,153.497
C03092=1082.311,55.882,-62.432,174.309,20.821,153.497
C03093=1082.317,56.131,-62.448,174.310,20.823,153.497
C03094=1082.322,56.381,-62.465,174.312,20.825,153.497
C03095=1082.328,56.630,-62.481,174.314,20.827,153.497
C03096=1082.334,56.880,-62.497,174.316,20.830,153.498
C03097=1082.340,57.129,-62.514,174.317,20.832,153.498
C03098=1082.346,57.378,-62.530,174.318,20.834,153.498
C03099=1082.351,57.628,-62.547,174.321,20.836,153.498
C03100=1082.357,57.877,-62.563,174.322,20.838,153.498
C03101=1082.363,58.127,-62.579,174.323,20.840,153.498
C03102=1082.369,58.376,-62.596,174.325,20.842,153.498
C03103=1082.375,58.625,-62.612,174.327,20.844,153.499
C03104=1082.380,58.875,-62.629,174.329,20.847,153.499
C03105=1082.386,59.124,-62.645,174.330,20.849,153.499
C03106=1082.392,59.374,-62.661,174.331,20.851,153.499
C03107=1082.398,59.623,-62.677,174.333,20.854,153.499
C03108=1082.404,59.872,-62.694,174.335,20.856,153.500
C03109=1082.409,60.122,-62.711,174.337,20.858,153.500
C03110=1082.415,60.371,-62.727,174.338,20.860,153.500
C03111=1082.421,60.621,-62.743,174.339,20.862,153.500
C03112=1082.427,60.870,-62.759,174.342,20.864,153.500
C03113=1082.432,61.120,-62.776,174.343,20.866,153.500
C03114=1082.438,61.369,-62.792,174.344,20.868,153.501
C03115=1082.444,61.618,-62.809,174.346,20.871,153.501
C03116=1082.450,61.867,-62.826,174.348,20.873,153.501
C03117=1082.455,62.106,-62.841,174.350,20.875,153.501
C03118=1082.462,62.344,-62.857,174.351,20.877,153.501
C03119=1082.467,62.583,-62.873,174.353,20.879,153.501
C03120=1082.473,62.820,-62.889,174.354,20.880,153.501
C03121=1082.478,63.059,-62.905,174.356,20.883,153.502
C03122=1082.484,63.297,-62.921,174.358,20.885,153.502
C03123=1082.489,63.536,-62.936,174.359,20.887,153.502
C03124=1082.495,63.773,-62.952,174.361,20.889,153.502
C03125=1082.501,64.024,-62.969,174.362,20.891,153.502
C03126=1082.507,64.273,-62.985,174.364,20.893,153.502
C03127=1082.513,64.523,-63.002,174.366,20.896,153.503
C03128=1082.518,64.772,-63.019,174.367,20.898,153.503
C03129=1082.524,65.021,-63.036,174.369,20.899,153.503
C03130=1082.529,65.271,-63.052,174.371,20.902,153.503
C03131=1082.535,65.520,-63.069,174.372,20.904,153.503
C03132=1082.541,65.769,-63.086,174.374,20.906,153.503
C03133=1082.547,66.018,-63.102,174.376,20.908,153.503
C03134=1082.553,66.268,-63.119,174.378,20.911,153.504
C03135=1082.558,66.517,-63.136,174.379,20.913,153.504
C03136=1082.564,66.766,-63.153,174.380,20.915,153.504
C03137=1082.569,67.016,-63.169,174.382,20.917,153.504
C03138=1082.575,67.265,-63.186,174.384,20.919,153.504
C03139=1082.582,67.515,-63.204,174.386,20.921,153.504
C03140=1082.587,67.764,-63.220,174.387,20.923,153.505
C03141=1082.593,68.014,-63.237,174.389,20.925,153.505
C03142=1082.599,68.263,-63.254,174.391,20.928,153.505
C03143=1082.604,68.512,-63.271,174.392,20.930,153.505
C03144=1082.610,68.762,-63.287,174.394,20.933,153.505
C03145=1082.616,69.011,-63.304,174.395,20.935,153.506
C03146=1082.621,69.260,-63.321,174.397,20.937,153.506
C03147=1082.627,69.510,-63.337,174.399,20.939,153.506
C03148=1082.632,69.759,-63.355,174.400,20.941,153.506
C03149=1082.639,70.009,-63.372,174.402,20.943,153.506
C03150=1082.644,70.258,-63.389,174.404,20.945,153.506
C03151=1082.650,70.507,-63.405,174.406,20.948,153.506
C03152=1082.656,70.757,-63.422,174.407,20.950,153.507
C03153=1082.661,71.006,-63.440,174.409,20.952,153.507
C03154=1082.667,71.255,-63.456,174.411,20.954,153.507
C03155=1082.673,71.504,-63.474,174.412,20.956,153.507
C03156=1082.678,71.754,-63.491,174.414,20.958,153.507
C03157=1082.685,72.003,-63.508,174.416,20.960,153.507
C03158=1082.690,72.253,-63.525,174.417,20.962,153.508
C03159=1082.695,72.502,-63.542,174.419,20.965,153.508
C03160=1082.701,72.751,-63.559,174.420,20.967,153.508
C03161=1082.707,73.000,-63.576,174.423,20.969,153.508
C03162=1082.712,73.250,-63.593,174.424,20.971,153.508
C03163=1082.718,73.499,-63.610,174.426,20.974,153.508
C03164=1082.724,73.749,-63.627,174.427,20.975,153.509
C03165=1082.730,73.998,-63.645,174.429,20.977,153.509
C03166=1082.736,74.247,-63.661,174.431,20.980,153.509
C03167=1082.741,74.496,-63.679,174.432,20.982,153.509
C03168=1082.746,74.746,-63.695,174.434,20.984,153.509
C03169=1082.753,74.995,-63.712,174.436,20.986,153.509
C03170=1082.758,75.245,-63.730,174.438,20.989,153.509
C03171=1082.764,75.494,-63.747,174.439,20.990,153.510
C03172=1082.769,75.743,-63.765,174.441,20.992,153.510
C03173=1082.775,75.993,-63.781,174.443,20.994,153.510
C03174=1082.781,76.242,-63.799,174.444,20.996,153.510
C03175=1082.787,76.492,-63.816,174.446,20.999,153.510
C03176=1082.793,76.741,-63.833,174.448,21.001,153.510
C03177=1082.798,76.990,-63.850,174.450,21.003,153.510
C03178=1082.804,77.240,-63.867,174.451,21.005,153.511
C03179=1082.809,77.489,-63.885,174.453,21.008,153.511
C03180=1082.816,77.738,-63.902,174.455,21.009,153.511
C03181=1082.821,77.988,-63.919,174.456,21.011,153.511
C03182=1082.827,78.237,-63.937,174.458,21.014,153.511
C03183=1082.832,78.486,-63.954,174.460,21.016,153.511
C03184=1082.838,78.736,-63.971,174.462,21.018,153.512
C03185=1082.844,79.015,-63.991,174.463,21.020,153.512
C03186=1082.851,79.294,-64.011,174.465,21.023,153.512
C03187=1082.857,79.574,-64.030,174.467,21.025,153.512
C03188=1082.863,79.852,-64.049,174.470,21.027,153.512
C03189=1082.869,80.101,-64.067,174.471,21.029,153.512
C03190=1082.875,80.352,-64.084,174.473,21.032,153.512
C03191=1082.880,80.601,-64.101,174.474,21.034,153.513
C03192=1082.886,80.849,-64.118,174.477,21.036,153.513
C03193=1082.892,81.098,-64.136,174.478,21.038,153.513
C03194=1082.898,81.349,-64.153,174.479,21.040,153.513
C03195=1082.903,81.598,-64.171,174.481,21.042,153.513
C03196=1082.909,81.847,-64.188,174.483,21.044,153.513
C03197=1082.914,82.096,-64.206,174.485,21.047,153.514
C03198=1082.920,82.346,-64.224,174.486,21.049,153.514
C03199=1082.926,82.595,-64.241,174.488,21.051,153.514
C03200=1082.931,82.844,-64.258,174.490,21.053,153.514
C03201=1082.937,83.093,-64.276,174.492,21.056,153.514
C03202=1082.943,83.343,-64.294,174.493,21.058,153.514
C03203=1082.948,83.592,-64.311,174.495,21.060,153.515
C03204=1082.954,83.841,-64.329,174.497,21.061,153.515
C03205=1082.960,84.091,-64.347,174.499,21.064,153.515
C03206=1082.965,84.341,-64.364,174.501,21.066,153.515
C03207=1082.971,84.590,-64.381,174.502,21.068,153.515
C03208=1082.976,84.839,-64.399,174.504,21.070,153.515
C03209=1082.982,85.088,-64.417,174.505,21.072,153.515
C03210=1082.988,85.337,-64.434,174.508,21.074,153.516
C03211=1082.993,85.587,-64.452,174.509,21.076,153.516
C03212=1082.999,85.836,-64.470,174.511,21.078,153.516
C03213=1083.005,86.085,-64.487,174.513,21.080,153.516
C03214=1083.011,86.334,-64.505,174.515,21.083,153.516
C03215=1083.017,86.584,-64.523,174.516,21.085,153.516
C03216=1083.022,86.833,-64.540,174.518,21.087,153.516
C03217=1083.028,87.082,-64.558,174.520,21.089,153.517
C03218=1083.034,87.332,-64.576,174.522,21.091,153.517
C03219=1083.039,87.581,-64.593,174.523,21.093,153.517
C03220=1083.045,87.831,-64.611,174.526,21.095,153.517
C03221=1083.051,88.080,-64.629,174.527,21.097,153.517
C03222=1083.056,88.329,-64.646,174.529,21.100,153.517
C03223=1083.063,88.578,-64.664,174.530,21.102,153.517
C03224=1083.068,88.828,-64.682,174.532,21.103,153.517
C03225=1083.074,89.077,-64.700,174.534,21.105,153.518
C03226=1083.080,89.326,-64.717,174.535,21.107,153.518
C03227=1083.085,89.575,-64.735,174.538,21.110,153.518
C03228=1083.091,89.825,-64.753,174.539,21.112,153.518
C03229=1083.097,90.074,-64.771,174.541,21.114,153.518
C03230=1083.103,90.324,-64.788,174.543,21.116,153.518
C03231=1083.109,90.573,-64.806,174.545,21.118,153.518
C03232=1083.114,90.822,-64.824,174.546,21.120,153.519
C03233=1083.120,91.071,-64.843,174.549,21.122,153.519
C03234=1083.125,91.320,-64.860,174.550,21.124,153.519
C03235=1083.131,91.570,-64.878,174.552,21.126,153.519
C03236=1083.137,91.819,-64.896,174.553,21.128,153.519
C03237=1083.142,92.068,-64.914,174.556,21.130,153.519
C03238=1083.148,92.318,-64.932,174.557,21.132,153.519
C03239=1083.153,92.567,-64.950,174.559,21.134,153.519
C03240=1083.159,92.816,-64.968,174.561,21.136,153.520
C03241=1083.165,93.066,-64.986,174.563,21.139,153.520
C03242=1083.170,93.315,-65.004,174.564,21.141,153.520
C03243=1083.176,93.565,-65.022,174.566,21.143,153.520
C03244=1083.182,93.814,-65.039,174.568,21.145,153.520
C03245=1083.187,94.063,-65.059,174.570,21.147,153.520
C03246=1083.193,94.312,-65.076,174.571,21.149,153.520
C03247=1083.198,94.561,-65.094,174.574,21.151,153.520
C03248=1083.205,94.811,-65.112,174.575,21.153,153.521
C03249=1083.211,95.090,-65.133,174.577,21.156,153.521
C03250=1083.217,95.369,-65.153,174.579,21.158,153.521
C03251=1083.223,95.649,-65.173,174.582,21.160,153.521
C03252=1083.229,95.928,-65.193,174.584,21.163,153.521
C03253=1083.235,96.177,-65.212,174.585,21.164,153.521
C03254=1083.241,96.426,-65.230,174.588,21.167,153.521
C03255=1083.247,96.675,-65.247,174.589,21.169,153.522
C03256=1083.252,96.925,-65.266,174.591,21.171,153.522
C03257=1083.258,97.174,-65.284,174.593,21.172,153.522
C03258=1083.264,97.424,-65.302,174.595,21.175,153.522
C03259=1083.269,97.673,-65.320,174.596,21.177,153.522
C03260=1083.275,97.922,-65.339,174.598,21.179,153.522
C03261=1083.281,98.171,-65.356,174.600,21.181,153.522
C03262=1083.287,98.420,-65.376,174.602,21.183,153.522
C03263=1083.292,98.670,-65.393,174.603,21.185,153.523
C03264=1083.298,98.919,-65.411,174.606,21.187,153.523
C03265=1083.303,99.168,-65.430,174.607,21.189,153.523
C03266=1083.309,99.418,-65.448,174.609,21.191,153.523
C03267=1083.315,99.666,-65.466,174.611,21.193,153.523
C03268=1083.321,99.916,-65.485,174.613,21.195,153.523
C03269=1083.326,100.165,-65.502,174.614,21.197,153.523
C03270=1083.333,100.414,-65.521,174.617,21.199,153.523
C03271=1083.337,100.664,-65.539,174.618,21.201,153.523
C03272=1083.344,100.913,-65.558,174.620,21.203,153.524
C03273=1083.350,101.163,-65.576,174.622,21.205,153.524
C03274=1083.355,101.411,-65.595,174.624,21.207,153.524
C03275=1083.361,101.661,-65.612,174.625,21.209,153.524
C03276=1083.366,101.910,-65.631,174.628,21.211,153.524
C03277=1083.372,102.160,-65.650,174.630,21.213,153.524
C03278=1083.377,102.408,-65.668,174.631,21.215,153.524
C03279=1083.383,102.658,-65.687,174.634,21.218,153.524
C03280=1083.389,102.907,-65.705,174.635,21.220,153.525
C03281=1083.394,103.157,-65.723,174.637,21.221,153.525
C03282=1083.400,103.405,-65.742,174.639,21.223,153.525
C03283=1083.405,103.655,-65.760,174.641,21.226,153.525
C03284=1083.411,103.904,-65.779,174.642,21.227,153.525
C03285=1083.417,104.153,-65.798,174.645,21.230,153.525
C03286=1083.423,104.403,-65.816,174.646,21.232,153.525
C03287=1083.428,104.652,-65.835,174.648,21.233,153.525
C03288=1083.433,104.902,-65.853,174.650,21.235,153.525
C03289=1083.439,105.150,-65.871,174.652,21.238,153.526
C03290=1083.445,105.400,-65.891,174.654,21.240,153.526
C03291=1083.450,105.649,-65.908,174.656,21.242,153.526
C03292=1083.456,105.898,-65.928,174.658,21.244,153.526
C03293=1083.461,106.148,-65.946,174.659,21.245,153.526
C03294=1083.467,106.396,-65.964,174.661,21.248,153.526
C03295=1083.473,106.646,-65.984,174.663,21.250,153.526
C03296=1083.479,106.896,-66.001,174.665,21.252,153.526
C03297=1083.484,107.144,-66.020,174.667,21.254,153.526
C03298=1083.490,107.394,-66.040,174.669,21.256,153.527
C03299=1083.496,107.642,-66.058,174.671,21.258,153.527
C03300=1083.501,107.892,-66.076,174.672,21.260,153.527
C03301=1083.507,108.141,-66.095,174.675,21.262,153.527
C03302=1083.513,108.390,-66.114,174.676,21.264,153.527
C03303=1083.518,108.640,-66.132,174.678,21.266,153.527
C03304=1083.524,108.889,-66.151,174.680,21.267,153.527
C03305=1083.529,109.138,-66.170,174.682,21.270,153.527
C03306=1083.536,109.387,-66.189,174.684,21.271,153.527
C03307=1083.541,109.637,-66.207,174.686,21.274,153.527
C03308=1083.546,109.886,-66.226,174.688,21.276,153.527
C03309=1083.553,110.135,-66.245,174.690,21.277,153.528
C03310=1083.558,110.384,-66.264,174.692,21.280,153.528
C03311=1083.563,110.633,-66.283,174.693,21.281,153.528
C03312=1083.570,110.883,-66.301,174.696,21.284,153.528
C03313=1083.576,111.162,-66.322,174.698,21.286,153.528
C03314=1083.583,111.442,-66.343,174.700,21.288,153.528
C03315=1083.589,111.720,-66.364,174.702,21.290,153.528
C03316=1083.595,111.999,-66.386,174.704,21.292,153.528
C03317=1083.601,112.249,-66.405,174.706,21.294,153.528
C03318=1083.606,112.499,-66.423,174.708,21.296,153.529
C03319=1083.612,112.748,-66.443,174.710,21.298,153.529
C03320=1083.617,112.997,-66.461,174.712,21.300,153.529
C03321=1083.623,113.246,-66.480,174.714,21.302,153.529
C03322=1083.629,113.496,-66.499,174.716,21.304,153.529
C03323=1083.634,113.744,-66.518,174.717,21.306,153.529
C03324=1083.640,113.994,-66.537,174.720,21.308,153.529
C03325=1083.646,114.243,-66.556,174.722,21.310,153.529
C03326=1083.652,114.492,-66.575,174.723,21.312,153.529
C03327=1083.657,114.741,-66.594,174.726,21.314,153.529
C03328=1083.663,114.990,-66.613,174.727,21.316,153.529
C03329=1083.668,115.240,-66.633,174.729,21.318,153.530
C03330=1083.674,115.489,-66.652,174.731,21.320,153.530
C03331=1083.679,115.738,-66.671,174.733,21.322,153.530
C03332=1083.685,115.987,-66.690,174.735,21.324,153.530
C03333=1083.690,116.236,-66.709,174.737,21.326,153.530
C03334=1083.696,116.486,-66.728,174.739,21.328,153.530
C03335=1083.701,116.735,-66.747,174.740,21.330,153.530
C03336=1083.707,116.984,-66.766,174.743,21.332,153.530
C03337=1083.712,117.233,-66.786,174.745,21.334,153.530
C03338=1083.718,117.483,-66.805,174.747,21.336,153.531
C03339=1083.724,117.732,-66.824,174.749,21.338,153.531
C03340=1083.729,117.981,-66.843,174.750,21.340,153.531
C03341=1083.734,118.230,-66.862,174.752,21.342,153.531
C03342=1083.740,118.480,-66.881,174.755,21.344,153.531
C03343=1083.746,118.729,-66.901,174.756,21.346,153.531
C03344=1083.751,118.978,-66.920,174.758,21.348,153.531
C03345=1083.757,119.227,-66.939,174.760,21.350,153.531
C03346=1083.762,119.476,-66.959,174.762,21.352,153.531
C03347=1083.768,119.726,-66.978,174.765,21.354,153.531
C03348=1083.773,119.974,-66.997,174.766,21.356,153.532
C03349=1083.779,120.224,-67.016,174.768,21.358,153.532
C03350=1083.785,120.473,-67.035,174.771,21.360,153.532
C03351=1083.790,120.723,-67.055,174.772,21.361,153.532
C03352=1083.796,120.971,-67.075,174.774,21.364,153.532
C03353=1083.801,121.220,-67.093,174.776,21.365,153.532
C03354=1083.807,121.470,-67.113,174.778,21.368,153.532
C03355=1083.813,121.719,-67.132,174.781,21.370,153.532
C03356=1083.818,121.968,-67.151,174.782,21.371,153.532
C03357=1083.824,122.217,-67.171,174.784,21.373,153.532
C03358=1083.829,122.467,-67.191,174.786,21.375,153.532
C03359=1083.835,122.716,-67.210,174.788,21.377,153.532
C03360=1083.840,122.965,-67.229,174.790,21.379,153.532
C03361=1083.846,123.214,-67.249,174.792,21.381,153.533
C03362=1083.852,123.463,-67.268,174.794,21.383,153.533
C03363=1083.858,123.713,-67.287,174.796,21.385,153.533
C03364=1083.864,123.962,-67.307,174.798,21.387,153.533
C03365=1083.869,124.210,-67.326,174.800,21.388,153.533
C03366=1083.874,124.460,-67.346,174.803,21.391,153.533
C03367=1083.880,124.709,-67.366,174.804,21.392,153.533
C03368=1083.886,124.958,-67.385,174.806,21.395,153.533
C03369=1083.892,125.207,-67.404,174.808,21.396,153.533
C03370=1083.897,125.457,-67.425,174.810,21.398,153.533
C03371=1083.903,125.706,-67.444,174.812,21.400,153.533
C03372=1083.908,125.955,-67.463,174.814,21.402,153.533
C03373=1083.914,126.204,-67.483,174.816,21.404,153.533
C03374=1083.920,126.454,-67.502,174.819,21.406,153.534
C03375=1083.925,126.702,-67.521,174.820,21.407,153.534
C03376=1083.931,126.951,-67.541,174.823,21.409,153.534
C03377=1083.937,127.231,-67.563,174.825,21.412,153.534
C03378=1083.944,127.510,-67.585,174.827,21.414,153.534
C03379=1083.950,127.789,-67.607,174.829,21.416,153.534
C03380=1083.957,128.068,-67.629,174.832,21.418,153.534
C03381=1083.962,128.318,-67.649,174.833,21.420,153.534
C03382=1083.968,128.567,-67.669,174.836,21.422,153.534
C03383=1083.974,128.816,-67.688,174.838,21.424,153.534
C03384=1083.980,129.065,-67.708,174.839,21.425,153.534
C03385=1083.985,129.315,-67.727,174.842,21.427,153.534
C03386=1083.991,129.563,-67.747,174.844,21.429,153.534
C03387=1083.997,129.813,-67.767,174.846,21.431,153.534
C03388=1084.002,130.062,-67.787,174.848,21.433,153.534
C03389=1084.008,130.311,-67.806,174.850,21.435,153.534
C03390=1084.014,130.560,-67.826,174.852,21.436,153.535
C03391=1084.020,130.810,-67.846,174.854,21.439,153.535
C03392=1084.026,131.059,-67.866,174.857,21.441,153.535
C03393=1084.031,131.308,-67.885,174.858,21.442,153.535
C03394=1084.037,131.557,-67.905,174.861,21.444,153.535
C03395=1084.043,131.806,-67.925,174.863,21.446,153.535
C03396=1084.048,132.055,-67.945,174.864,21.448,153.535
C03397=1084.054,132.304,-67.965,174.867,21.450,153.535
C03398=1084.059,132.554,-67.984,174.869,21.451,153.535
C03399=1084.065,132.803,-68.004,174.871,21.453,153.535
C03400=1084.070,133.052,-68.025,174.873,21.455,153.535
C03401=1084.076,133.301,-68.044,174.875,21.457,153.535
C03402=1084.082,133.550,-68.064,174.877,21.459,153.535
C03403=1084.087,133.799,-68.085,174.879,21.461,153.535
C03404=1084.093,134.049,-68.104,174.882,21.463,153.535
C03405=1084.098,134.298,-68.124,174.883,21.465,153.536
C03406=1084.104,134.547,-68.144,174.885,21.467,153.536
C03407=1084.109,134.796,-68.164,174.888,21.468,153.536
C03408=1084.115,135.045,-68.184,174.889,21.470,153.536
C03409=1084.121,135.294,-68.204,174.891,21.472,153.536
C03410=1084.127,135.543,-68.225,174.894,21.474,153.536
C03411=1084.132,135.792,-68.244,174.895,21.476,153.536
C03412=1084.137,136.042,-68.265,174.898,21.478,153.536
C03413=1084.143,136.290,-68.284,174.900,21.480,153.536
C03414=1084.149,136.540,-68.305,174.903,21.482,153.536
C03415=1084.154,136.789,-68.324,174.904,21.483,153.536
C03416=1084.160,137.038,-68.344,174.906,21.485,153.536
C03417=1084.166,137.287,-68.365,174.909,21.487,153.536
C03418=1084.172,137.536,-68.385,174.910,21.489,153.536
C03419=1084.177,137.785,-68.405,174.913,21.491,153.536
C03420=1084.183,138.034,-68.426,174.915,21.493,153.536
C03421=1084.188,138.284,-68.445,174.916,21.494,153.536
C03422=1084.194,138.533,-68.465,174.919,21.496,153.536
C03423=1084.200,138.782,-68.486,174.921,21.498,153.536
C03424=1084.206,139.031,-68.506,174.923,21.500,153.537
C03425=1084.211,139.280,-68.527,174.925,21.502,153.537
C03426=1084.217,139.529,-68.546,174.927,21.504,153.537
C03427=1084.222,139.778,-68.567,174.930,21.506,153.537
C03428=1084.227,140.027,-68.588,174.931,21.507,153.537
C03429=1084.233,140.276,-68.607,174.934,21.509,153.537
C03430=1084.238,140.526,-68.627,174.936,21.511,153.537
C03431=1084.245,140.775,-68.648,174.938,21.513,153.537
C03432=1084.250,141.024,-68.668,174.940,21.515,153.537
C03433=1084.255,141.273,-68.689,174.942,21.516,153.537
C03434=1084.261,141.522,-68.709,174.945,21.519,153.537
C03435=1084.267,141.771,-68.729,174.946,21.520,153.537
C03436=1084.273,142.020,-68.749,174.949,21.522,153.537
C03437=1084.278,142.269,-68.770,174.951,21.524,153.537
C03438=1084.283,142.518,-68.790,174.953,21.526,153.537
C03439=1084.289,142.767,-68.810,174.955,21.528,153.537
C03440=1084.295,143.017,-68.831,174.957,21.530,153.537
C03441=1084.301,143.296,-68.854,174.960,21.532,153.537
C03442=1084.307,143.575,-68.876,174.962,21.534,153.537
C03443=1084.313,143.854,-68.901,174.964,21.536,153.537
C03444=1084.320,144.133,-68.923,174.967,21.538,153.537
C03445=1084.326,144.382,-68.943,174.969,21.539,153.537
C03446=1084.331,144.631,-68.964,174.971,21.542,153.538
C03447=1084.336,144.880,-68.984,174.974,21.544,153.538
C03448=1084.343,145.130,-69.005,174.975,21.545,153.538
C03449=1084.348,145.379,-69.025,174.978,21.547,153.538
C03450=1084.353,145.628,-69.046,174.980,21.549,153.538
C03451=1084.359,145.877,-69.067,174.982,21.550,153.538
C03452=1084.365,146.125,-69.087,174.984,21.552,153.538
C03453=1084.371,146.375,-69.108,174.986,21.555,153.538
C03454=1084.376,146.624,-69.129,174.989,21.556,153.538
C03455=1084.381,146.873,-69.149,174.990,21.558,153.538
C03456=1084.387,147.122,-69.169,174.993,21.560,153.538
C03457=1084.393,147.371,-69.191,174.995,21.562,153.538
C03458=1084.399,147.621,-69.211,174.998,21.563,153.538
C03459=1084.405,147.869,-69.231,174.999,21.565,153.538
C03460=1084.410,148.119,-69.252,175.002,21.567,153.538
C03461=1084.415,148.368,-69.272,175.004,21.569,153.538
C03462=1084.421,148.617,-69.294,175.006,21.571,153.538
C03463=1084.427,148.866,-69.314,175.009,21.573,153.538
C03464=1084.432,149.115,-69.335,175.010,21.574,153.538
C03465=1084.438,149.364,-69.355,175.013,21.576,153.538
C03466=1084.444,149.613,-69.377,175.015,21.578,153.538
C03467=1084.449,149.862,-69.397,175.018,21.580,153.538
C03468=1084.455,150.111,-69.418,175.019,21.581,153.538
C03469=1084.460,150.360,-69.439,175.022,21.583,153.538
C03470=1084.466,150.610,-69.460,175.024,21.585,153.538
C03471=1084.471,150.859,-69.480,175.026,21.587,153.539
C03472=1084.477,151.107,-69.502,175.028,21.589,153.539
C03473=1084.482,151.356,-69.522,175.030,21.591,153.539
C03474=1084.488,151.606,-69.543,175.033,21.592,153.539
C03475=1084.494,151.854,-69.564,175.035,21.594,153.539
C03476=1084.499,152.104,-69.584,175.037,21.596,153.539
C03477=1084.505,152.353,-69.605,175.039,21.598,153.539
C03478=1084.511,152.602,-69.627,175.041,21.599,153.539
C03479=1084.516,152.851,-69.647,175.044,21.601,153.539
C03480=1084.522,153.100,-69.668,175.046,21.603,153.539
C03481=1084.528,153.349,-69.689,175.048,21.605,153.539
C03482=1084.533,153.598,-69.711,175.050,21.607,153.539
C03483=1084.538,153.847,-69.731,175.052,21.609,153.539
C03484=1084.544,154.097,-69.752,175.055,21.611,153.539
C03485=1084.550,154.345,-69.773,175.057,21.613,153.539
C03486=1084.555,154.594,-69.794,175.059,21.614,153.539
C03487=1084.561,154.844,-69.816,175.061,21.616,153.539
C03488=1084.566,155.093,-69.836,175.064,21.618,153.539
C03489=1084.572,155.341,-69.857,175.066,21.620,153.539
C03490=1084.578,155.591,-69.878,175.069,21.621,153.539
C03491=1084.583,155.840,-69.900,175.070,21.623,153.539
C03492=1084.589,156.088,-69.921,175.073,21.625,153.539
C03493=1084.595,156.338,-69.942,175.075,21.627,153.539
C03494=1084.600,156.586,-69.963,175.077,21.628,153.539
C03495=1084.606,156.836,-69.984,175.080,21.630,153.539
C03496=1084.611,157.085,-70.006,175.081,21.632,153.539
C03497=1084.616,157.334,-70.026,175.084,21.634,153.539
C03498=1084.622,157.583,-70.048,175.086,21.635,153.539
C03499=1084.628,157.832,-70.069,175.089,21.637,153.539
C03500=1084.633,158.081,-70.090,175.091,21.639,153.539
C03501=1084.639,158.330,-70.111,175.094,21.641,153.539
C03502=1084.645,158.579,-70.132,175.095,21.642,153.539
C03503=1084.650,158.828,-70.153,175.097,21.644,153.539
C03504=1084.656,159.077,-70.175,175.100,21.646,153.539
C03505=1084.662,159.356,-70.199,175.102,21.648,153.539
C03506=1084.668,159.635,-70.223,175.105,21.650,153.539
C03507=1084.675,159.914,-70.247,175.107,21.652,153.539
C03508=1084.681,160.193,-70.271,175.110,21.655,153.539
C03509=1084.686,160.442,-70.291,175.112,21.656,153.539
C03510=1084.693,160.691,-70.313,175.114,21.657,153.539
C03511=1084.698,160.940,-70.334,175.117,21.659,153.539
C03512=1084.704,161.188,-70.355,175.119,21.661,153.539
C03513=1084.709,161.438,-70.377,175.122,21.663,153.539
C03514=1084.714,161.687,-70.398,175.124,21.665,153.539
C03515=1084.720,161.936,-70.420,175.127,21.667,153.539
C03516=1084.725,162.185,-70.442,175.128,21.669,153.540
C03517=1084.731,162.434,-70.462,175.130,21.670,153.540
C03518=1084.736,162.683,-70.484,175.133,21.672,153.540
C03519=1084.742,162.932,-70.506,175.135,21.674,153.540
C03520=1084.748,163.181,-70.527,175.138,21.676,153.540
C03521=1084.753,163.430,-70.549,175.140,21.678,153.540
C03522=1084.758,163.678,-70.571,175.142,21.679,153.540
C03523=1084.763,163.929,-70.592,175.144,21.681,153.540
C03524=1084.769,164.177,-70.613,175.147,21.683,153.540
C03525=1084.774,164.426,-70.635,175.149,21.685,153.540
C03526=1084.780,164.675,-70.657,175.151,21.687,153.540
C03527=1084.785,164.924,-70.679,175.154,21.689,153.540
C03528=1084.791,165.173,-70.700,175.156,21.690,153.540
C03529=1084.796,165.422,-70.722,175.158,21.692,153.540
C03530=1084.802,165.671,-70.744,175.160,21.694,153.540
C03531=1084.807,165.920,-70.765,175.163,21.696,153.540
C03532=1084.813,166.169,-70.787,175.165,21.697,153.540
C03533=1084.818,166.418,-70.809,175.167,21.700,153.540
C03534=1084.823,166.667,-70.830,175.170,21.702,153.540
C03535=1084.829,166.916,-70.851,175.172,21.703,153.540
C03536=1084.834,167.165,-70.873,175.175,21.705,153.540
C03537=1084.840,167.414,-70.895,175.176,21.707,153.540
C03538=1084.845,167.663,-70.917,175.179,21.708,153.540
C03539=1084.851,167.912,-70.938,175.181,21.710,153.540
C03540=1084.856,168.161,-70.961,175.184,21.712,153.540
C03541=1084.862,168.410,-70.983,175.186,21.714,153.540
C03542=1084.867,168.659,-71.004,175.189,21.716,153.540
C03543=1084.873,168.908,-71.026,175.191,21.717,153.540
C03544=1084.878,169.157,-71.048,175.193,21.719,153.540
C03545=1084.884,169.406,-71.070,175.196,21.721,153.540
C03546=1084.889,169.655,-71.091,175.197,21.722,153.540
C03547=1084.895,169.904,-71.113,175.200,21.724,153.540
C03548=1084.900,170.153,-71.135,175.202,21.726,153.540
C03549=1084.906,170.402,-71.157,175.205,21.728,153.540
C03550=1084.912,170.651,-71.179,175.207,21.730,153.540
C03551=1084.917,170.900,-71.201,175.210,21.732,153.540
C03552=1084.923,171.149,-71.223,175.212,21.734,153.540
C03553=1084.928,171.398,-71.245,175.214,21.735,153.540
C03554=1084.934,171.647,-71.267,175.217,21.737,153.540
C03555=1084.939,171.896,-71.288,175.219,21.739,153.540
C03556=1084.945,172.145,-71.310,175.221,21.740,153.540
C03557=1084.951,172.394,-71.333,175.223,21.742,153.540
C03558=1084.955,172.643,-71.355,175.226,21.744,153.540
C03559=1084.962,172.892,-71.376,175.228,21.746,153.540
C03560=1084.966,173.141,-71.398,175.231,21.748,153.540
C03561=1084.973,173.389,-71.421,175.233,21.749,153.540
C03562=1084.978,173.639,-71.443,175.236,21.751,153.540
C03563=1084.984,173.887,-71.464,175.238,21.753,153.540
C03564=1084.989,174.137,-71.486,175.241,21.754,153.540
C03565=1084.995,174.386,-71.509,175.243,21.756,153.540
C03566=1085.001,174.634,-71.531,175.246,21.758,153.540
C03567=1085.006,174.884,-71.553,175.248,21.760,153.540
C03568=1085.012,175.132,-71.575,175.250,21.761,153.540
C03569=1085.018,175.412,-71.600,175.253,21.764,153.540
C03570=1085.024,175.690,-71.625,175.255,21.766,153.540
C03571=1085.030,175.968,-71.649,175.258,21.767,153.540
C03572=1085.037,176.247,-71.674,175.261,21.769,153.540
C03573=1085.043,176.496,-71.696,175.264,21.771,153.540
C03574=1085.048,176.744,-71.718,175.265,21.772,153.540
C03575=1085.053,176.994,-71.741,175.268,21.774,153.540
C03576=1085.060,177.242,-71.763,175.270,21.776,153.540
C03577=1085.065,177.491,-71.785,175.273,21.778,153.540
C03578=1085.070,177.740,-71.808,175.275,21.779,153.540
C03579=1085.077,177.989,-71.830,175.278,21.781,153.540
C03580=1085.082,178.239,-71.852,175.280,21.783,153.540
C03581=1085.087,178.487,-71.874,175.283,21.784,153.540
C03582=1085.093,178.736,-71.896,175.285,21.786,153.540
C03583=1085.099,178.985,-71.919,175.288,21.788,153.540
C03584=1085.104,179.234,-71.941,175.290,21.790,153.540
C03585=1085.110,179.482,-71.963,175.293,21.791,153.540
C03586=1085.116,179.732,-71.985,175.295,21.793,153.540
C03587=1085.121,179.981,-72.008,175.297,21.795,153.540
C03588=1085.128,180.230,-72.030,175.300,21.797,153.540
C03589=1085.133,180.479,-72.053,175.303,21.798,153.540
C03590=1085.138,180.727,-72.075,175.305,21.800,153.540
C03591=1085.145,180.976,-72.097,175.307,21.802,153.540
C03592=1085.150,181.225,-72.120,175.310,21.804,153.540
C03593=1085.156,181.475,-72.142,175.312,21.805,153.540
C03594=1085.161,181.724,-72.165,175.315,21.807,153.540
C03595=1085.167,181.971,-72.187,175.317,21.809,153.540
C03596=1085.173,182.221,-72.209,175.320,21.810,153.540
C03597=1085.178,182.470,-72.232,175.322,21.812,153.540
C03598=1085.184,182.719,-72.255,175.324,21.814,153.540
C03599=1085.190,182.968,-72.277,175.327,21.815,153.540
C03600=1085.196,183.217,-72.300,175.329,21.817,153.540
C03601=1085.201,183.466,-72.322,175.331,21.819,153.540
C03602=1085.207,183.715,-72.345,175.334,21.820,153.540
C03603=1085.213,183.963,-72.367,175.337,21.822,153.540
C03604=1085.219,184.212,-72.390,175.339,21.824,153.540
C03605=1085.224,184.462,-72.412,175.342,21.825,153.540
C03606=1085.230,184.710,-72.435,175.344,21.827,153.540
C03607=1085.236,184.959,-72.458,175.346,21.829,153.540
C03608=1085.242,185.208,-72.480,175.349,21.830,153.539
C03609=1085.247,185.457,-72.502,175.352,21.832,153.540
C03610=1085.252,185.706,-72.526,175.354,21.834,153.540
C03611=1085.258,185.955,-72.549,175.356,21.836,153.540
C03612=1085.264,186.204,-72.572,175.359,21.837,153.540
C03613=1085.268,186.453,-72.594,175.361,21.839,153.540
C03614=1085.274,186.701,-72.617,175.364,21.841,153.540
C03615=1085.280,186.950,-72.640,175.366,21.843,153.540
C03616=1085.286,187.199,-72.662,175.369,21.844,153.540
C03617=1085.291,187.448,-72.685,175.371,21.846,153.540
C03618=1085.296,187.697,-72.709,175.375,21.848,153.540
C03619=1085.301,187.946,-72.732,175.377,21.850,153.540
C03620=1085.307,188.195,-72.754,175.379,21.852,153.540
C03621=1085.313,188.444,-72.777,175.382,21.854,153.540
C03622=1085.318,188.693,-72.800,175.384,21.856,153.540
C03623=1085.323,188.941,-72.822,175.387,21.857,153.539
C03624=1085.328,189.190,-72.846,175.389,21.859,153.539
C03625=1085.334,189.439,-72.869,175.392,21.861,153.539
C03626=1085.340,189.688,-72.892,175.394,21.863,153.540
C03627=1085.346,189.937,-72.915,175.397,21.865,153.540
C03628=1085.351,190.186,-72.938,175.399,21.866,153.539
C03629=1085.357,190.435,-72.961,175.402,21.868,153.539
C03630=1085.361,190.683,-72.984,175.404,21.870,153.539
C03631=1085.367,190.932,-73.007,175.407,21.872,153.539
C03632=1085.373,191.181,-73.030,175.409,21.873,153.539
C03633=1085.379,191.459,-73.056,175.412,21.875,153.539
C03634=1085.386,191.738,-73.081,175.415,21.877,153.539
C03635=1085.391,192.016,-73.107,175.417,21.879,153.539
C03636=1085.397,192.294,-73.133,175.421,21.881,153.539
